LIN {X 0,Y 654.858,Z 275.472,A -85,B 0,C 180,E1 -5918.674,E2 -5918.674} C_VEL
LIN {X 0,Y 654.812,Z 275.476,A -85,B 0,C 180,E1 -5921.282,E2 -5921.282} C_VEL
LIN {X 0,Y 654.839,Z 275.478,A -85,B 0,C 180,E1 -5923.853,E2 -5923.853} C_VEL
LIN {X 0,Y 654.892,Z 275.466,A -85,B 0,C 180,E1 -5927.02,E2 -5927.02} C_VEL
LIN {X 0,Y 654.922,Z 275.602,A -85,B 0,C 180,E1 -5929.598,E2 -5929.598} C_VEL
LIN {X 0,Y 656.022,Z 282.75,A -85,B 0,C 180,E1 -5930.474,E2 -5930.474} C_VEL
LIN {X 0,Y 655.91,Z 303.676,A -85,B 0,C 180,E1 -5932.946,E2 -5932.946} C_VEL
LIN {X 0,Y 655.529,Z 325.625,A -85,B 0,C 180,E1 -5935.557,E2 -5935.557} C_VEL
LIN {X 0,Y 655.353,Z 341.331,A -85,B 0,C 180,E1 -5937.435,E2 -5937.435} C_VEL
LIN {X 0,Y 657.094,Z 353.746,A -85,B 0,C 180,E1 -5937.633,E2 -5937.633} C_VEL
LIN {X 0,Y 656.345,Z 478.954,A -85,B 0,C 180,E1 -5939.083,E2 -5939.083} C_VEL
LIN {X 0,Y 656.153,Z 493.285,A -85,B 0,C 180,E1 -5939.369,E2 -5939.369} C_VEL
LIN {X 0,Y 655.95,Z 507.048,A -85,B 0,C 180,E1 -5939.771,E2 -5939.771} C_VEL
LIN {X 0,Y 655.672,Z 519.008,A -85,B 0,C 180,E1 -5940.23,E2 -5940.23} C_VEL
LIN {X 0,Y 655.42,Z 531.637,A -85,B 0,C 180,E1 -5940.842,E2 -5940.842} C_VEL
LIN {X 0,Y 655.226,Z 543.124,A -85,B 0,C 180,E1 -5941.531,E2 -5941.531} C_VEL
LIN {X 0,Y 654.912,Z 553.719,A -85,B 0,C 180,E1 -5942.299,E2 -5942.299} C_VEL
LIN {X 0,Y 654.674,Z 564.21,A -85,B 0,C 180,E1 -5943.22,E2 -5943.22} C_VEL
LIN {X 0,Y 654.448,Z 572.913,A -85,B 0,C 180,E1 -5944.143,E2 -5944.143} C_VEL
LIN {X 0,Y 654.36,Z 581.161,A -85,B 0,C 180,E1 -5945.208,E2 -5945.208} C_VEL
LIN {X 0,Y 654.28,Z 587.098,A -85,B 0,C 180,E1 -5946.146,E2 -5946.146} C_VEL
LIN {X 0,Y 654.158,Z 593.341,A -85,B 0,C 180,E1 -5947.382,E2 -5947.382} C_VEL
LIN {X 0,Y 654.104,Z 597.95,A -85,B 0,C 180,E1 -5948.622,E2 -5948.622} C_VEL
LIN {X 0,Y 654.115,Z 601.066,A -85,B 0,C 180,E1 -5949.879,E2 -5949.879} C_VEL
LIN {X 0,Y 654.026,Z 602.743,A -85,B 0,C 180,E1 -5951.115,E2 -5951.115} C_VEL
LIN {X 0,Y 654.042,Z 603.068,A -85,B 0,C 180,E1 -5952.368,E2 -5952.368} C_VEL
LIN {X 0,Y 654.063,Z 602.012,A -85,B 0,C 180,E1 -5953.627,E2 -5953.627} C_VEL
LIN {X 0,Y 654.089,Z 599.535,A -85,B 0,C 180,E1 -5954.893,E2 -5954.893} C_VEL
LIN {X 0,Y 654.135,Z 596.647,A -85,B 0,C 180,E1 -5955.846,E2 -5955.846} C_VEL
LIN {X 0,Y 654.194,Z 591.408,A -85,B 0,C 180,E1 -5957.124,E2 -5957.124} C_VEL
LIN {X 0,Y 654.265,Z 586.234,A -85,B 0,C 180,E1 -5958.087,E2 -5958.087} C_VEL
LIN {X 0,Y 654.409,Z 578.75,A -85,B 0,C 180,E1 -5959.216,E2 -5959.216} C_VEL
LIN {X 0,Y 654.569,Z 570.797,A -85,B 0,C 180,E1 -5960.188,E2 -5960.188} C_VEL
LIN {X 0,Y 654.784,Z 561.084,A -85,B 0,C 180,E1 -5961.164,E2 -5961.164} C_VEL
LIN {X 0,Y 655.022,Z 550.211,A -85,B 0,C 180,E1 -5962.062,E2 -5962.062} C_VEL
LIN {X 0,Y 655.346,Z 538.21,A -85,B 0,C 180,E1 -5962.873,E2 -5962.873} C_VEL
LIN {X 0,Y 655.567,Z 526.146,A -85,B 0,C 180,E1 -5963.537,E2 -5963.537} C_VEL
LIN {X 0,Y 655.866,Z 513.079,A -85,B 0,C 180,E1 -5964.111,E2 -5964.111} C_VEL
LIN {X 0,Y 656.125,Z 499.646,A -85,B 0,C 180,E1 -5964.562,E2 -5964.562} C_VEL
LIN {X 0,Y 656.33,Z 485.485,A -85,B 0,C 180,E1 -5964.905,E2 -5964.905} C_VEL
LIN {X 0,Y 656.443,Z 470.534,A -85,B 0,C 180,E1 -5965.135,E2 -5965.135} C_VEL
LIN {X 0,Y 656.965,Z 351.438,A -85,B 0,C 180,E1 -5966.492,E2 -5966.492} C_VEL
LIN {X 0,Y 655.32,Z 341.034,A -85,B 0,C 180,E1 -5966.661,E2 -5966.661} C_VEL
LIN {X 0,Y 655.667,Z 317.93,A -85,B 0,C 180,E1 -5969.465,E2 -5969.465} C_VEL
LIN {X 0,Y 655.064,Z 314.605,A -85,B 0,C 180,E1 -5969.889,E2 -5969.889} C_VEL
LIN {X 0,Y 649.559,Z 304.313,A -85,B 0,C 180,E1 -5971.302,E2 -5971.302} C_VEL
LIN {X 0,Y 649.016,Z 300.937,A -85,B 0,C 180,E1 -5971.729,E2 -5971.729} C_VEL
LIN {X 0,Y 649.167,Z 283.958,A -85,B 0,C 180,E1 -5973.815,E2 -5973.815} C_VEL
LIN {X 0,Y 647.818,Z 276.352,A -85,B 0,C 180,E1 -5974.804,E2 -5974.804} C_VEL
LIN {X 0,Y 647.753,Z 276.352,A -85,B 0,C 180,E1 -5977.269,E2 -5977.269} C_VEL
LIN {X 0,Y 647.771,Z 276.354,A -85,B 0,C 180,E1 -5979.848,E2 -5979.848} C_VEL
LIN {X 0,Y 647.739,Z 276.355,A -85,B 0,C 180,E1 -5982.664,E2 -5982.664} C_VEL
LIN {X 0,Y 647.769,Z 276.352,A -85,B 0,C 180,E1 -5985.342,E2 -5985.342} C_VEL
LIN {X 0,Y 647.733,Z 276.357,A -85,B 0,C 180,E1 -5988.258,E2 -5988.258} C_VEL
LIN {X 0,Y 647.746,Z 276.354,A -85,B 0,C 180,E1 -5990.356,E2 -5990.356} C_VEL
LIN {X 0,Y 647.736,Z 276.355,A -85,B 0,C 180,E1 -5992.729,E2 -5992.729} C_VEL
LIN {X 0,Y 647.769,Z 276.356,A -85,B 0,C 180,E1 -5995.266,E2 -5995.266} C_VEL
LIN {X 0,Y 647.775,Z 276.35,A -85,B 0,C 180,E1 -5998.004,E2 -5998.004} C_VEL
LIN {X 0,Y 647.754,Z 276.353,A -85,B 0,C 180,E1 -6000.17,E2 -6000.17} C_VEL
LIN {X 0,Y 647.796,Z 276.353,A -85,B 0,C 180,E1 -6002.99,E2 -6002.99} C_VEL
LIN {X 0,Y 647.767,Z 276.351,A -85,B 0,C 180,E1 -6005.737,E2 -6005.737} C_VEL
LIN {X 0,Y 647.798,Z 276.353,A -85,B 0,C 180,E1 -6008.429,E2 -6008.429} C_VEL
LIN {X 0,Y 647.806,Z 276.348,A -85,B 0,C 180,E1 -6011.071,E2 -6011.071} C_VEL
LIN {X 0,Y 647.824,Z 276.344,A -85,B 0,C 180,E1 -6013.672,E2 -6013.672} C_VEL
LIN {X 0,Y 647.831,Z 276.35,A -85,B 0,C 180,E1 -6016.238,E2 -6016.238} C_VEL
LIN {X 0,Y 647.825,Z 276.343,A -85,B 0,C 180,E1 -6018.776,E2 -6018.776} C_VEL
LIN {X 0,Y 647.84,Z 276.343,A -85,B 0,C 180,E1 -6020.665,E2 -6020.665} C_VEL
LIN {X 0,Y 647.877,Z 276.339,A -85,B 0,C 180,E1 -6023.169,E2 -6023.169} C_VEL
LIN {X 0,Y 647.905,Z 276.391,A -85,B 0,C 180,E1 -6024.139,E2 -6024.139} C_VEL
LIN {X 0,Y 648.473,Z 281.744,A -85,B 0,C 180,E1 -6025.041,E2 -6025.041} C_VEL
LIN {X 0,Y 648.237,Z 295.521,A -85,B 0,C 180,E1 -6027.289,E2 -6027.289} C_VEL
LIN {X 0,Y 650.27,Z 305.689,A -85,B 0,C 180,E1 -6027.452,E2 -6027.452} C_VEL
LIN {X 0,Y 649.684,Z 431.042,A -85,B 0,C 180,E1 -6028.86,E2 -6028.86} C_VEL
LIN {X 0,Y 649.542,Z 445.303,A -85,B 0,C 180,E1 -6029.149,E2 -6029.149} C_VEL
LIN {X 0,Y 649.298,Z 459.578,A -85,B 0,C 180,E1 -6029.574,E2 -6029.574} C_VEL
LIN {X 0,Y 649.028,Z 472.244,A -85,B 0,C 180,E1 -6030.076,E2 -6030.076} C_VEL
LIN {X 0,Y 648.791,Z 484.553,A -85,B 0,C 180,E1 -6030.694,E2 -6030.694} C_VEL
LIN {X 0,Y 648.467,Z 495.848,A -85,B 0,C 180,E1 -6031.391,E2 -6031.391} C_VEL
LIN {X 0,Y 648.173,Z 506.232,A -85,B 0,C 180,E1 -6032.166,E2 -6032.166} C_VEL
LIN {X 0,Y 647.846,Z 516.572,A -85,B 0,C 180,E1 -6033.097,E2 -6033.097} C_VEL
LIN {X 0,Y 647.639,Z 525.114,A -85,B 0,C 180,E1 -6034.03,E2 -6034.03} C_VEL
LIN {X 0,Y 647.441,Z 533.416,A -85,B 0,C 180,E1 -6035.13,E2 -6035.13} C_VEL
LIN {X 0,Y 647.289,Z 539.975,A -85,B 0,C 180,E1 -6036.211,E2 -6036.211} C_VEL
LIN {X 0,Y 647.229,Z 544.542,A -85,B 0,C 180,E1 -6037.148,E2 -6037.148} C_VEL
LIN {X 0,Y 647.111,Z 548.238,A -85,B 0,C 180,E1 -6038.088,E2 -6038.088} C_VEL
LIN {X 0,Y 647.087,Z 551.85,A -85,B 0,C 180,E1 -6039.343,E2 -6039.343} C_VEL
LIN {X 0,Y 647.054,Z 554.075,A -85,B 0,C 180,E1 -6040.603,E2 -6040.603} C_VEL
LIN {X 0,Y 647.018,Z 554.949,A -85,B 0,C 180,E1 -6041.868,E2 -6041.868} C_VEL
LIN {X 0,Y 647.077,Z 554.469,A -85,B 0,C 180,E1 -6043.138,E2 -6043.138} C_VEL
LIN {X 0,Y 647.031,Z 552.613,A -85,B 0,C 180,E1 -6044.416,E2 -6044.416} C_VEL
LIN {X 0,Y 647.168,Z 549.3,A -85,B 0,C 180,E1 -6045.697,E2 -6045.697} C_VEL
LIN {X 0,Y 647.223,Z 544.379,A -85,B 0,C 180,E1 -6046.988,E2 -6046.988} C_VEL
LIN {X 0,Y 647.321,Z 539.593,A -85,B 0,C 180,E1 -6047.956,E2 -6047.956} C_VEL
LIN {X 0,Y 647.492,Z 532.494,A -85,B 0,C 180,E1 -6049.099,E2 -6049.099} C_VEL
LIN {X 0,Y 647.659,Z 524.764,A -85,B 0,C 180,E1 -6050.11,E2 -6050.11} C_VEL
LIN {X 0,Y 647.94,Z 515.908,A -85,B 0,C 180,E1 -6051.064,E2 -6051.064} C_VEL
LIN {X 0,Y 648.218,Z 505.973,A -85,B 0,C 180,E1 -6051.952,E2 -6051.952} C_VEL
LIN {X 0,Y 648.537,Z 495.768,A -85,B 0,C 180,E1 -6052.711,E2 -6052.711} C_VEL
LIN {X 0,Y 648.837,Z 484.221,A -85,B 0,C 180,E1 -6053.421,E2 -6053.421} C_VEL
LIN {X 0,Y 649.077,Z 471.862,A -85,B 0,C 180,E1 -6054.038,E2 -6054.038} C_VEL
LIN {X 0,Y 649.355,Z 459.191,A -85,B 0,C 180,E1 -6054.536,E2 -6054.536} C_VEL
LIN {X 0,Y 649.544,Z 444.878,A -85,B 0,C 180,E1 -6054.958,E2 -6054.958} C_VEL
LIN {X 0,Y 649.693,Z 430.473,A -85,B 0,C 180,E1 -6055.245,E2 -6055.245} C_VEL
LIN {X 0,Y 650.21,Z 305.17,A -85,B 0,C 180,E1 -6056.654,E2 -6056.654} C_VEL
LIN {X 0,Y 648.261,Z 295.606,A -85,B 0,C 180,E1 -6056.827,E2 -6056.827} C_VEL
LIN {X 0,Y 648.558,Z 281.937,A -85,B 0,C 180,E1 -6059.076,E2 -6059.076} C_VEL
LIN {X 0,Y 647.813,Z 276.353,A -85,B 0,C 180,E1 -6060.056,E2 -6060.056} C_VEL
LIN {X 0,Y 647.739,Z 276.357,A -85,B 0,C 180,E1 -6062.728,E2 -6062.728} C_VEL
LIN {X 0,Y 647.75,Z 276.353,A -85,B 0,C 180,E1 -6064.965,E2 -6064.965} C_VEL
LIN {X 0,Y 647.742,Z 276.359,A -85,B 0,C 180,E1 -6067.871,E2 -6067.871} C_VEL
LIN {X 0,Y 647.74,Z 276.356,A -85,B 0,C 180,E1 -6070.45,E2 -6070.45} C_VEL
LIN {X 0,Y 647.728,Z 276.355,A -85,B 0,C 180,E1 -6072.94,E2 -6072.94} C_VEL
LIN {X 0,Y 647.745,Z 276.35,A -85,B 0,C 180,E1 -6075.533,E2 -6075.533} C_VEL
LIN {X 0,Y 647.762,Z 276.355,A -85,B 0,C 180,E1 -6078.252,E2 -6078.252} C_VEL
LIN {X 0,Y 647.755,Z 276.353,A -85,B 0,C 180,E1 -6080.358,E2 -6080.358} C_VEL
LIN {X 0,Y 647.746,Z 276.35,A -85,B 0,C 180,E1 -6083.146,E2 -6083.146} C_VEL
LIN {X 0,Y 647.747,Z 276.346,A -85,B 0,C 180,E1 -6085.264,E2 -6085.264} C_VEL
LIN {X 0,Y 647.752,Z 276.355,A -85,B 0,C 180,E1 -6088.004,E2 -6088.004} C_VEL
LIN {X 0,Y 647.789,Z 276.349,A -85,B 0,C 180,E1 -6090.172,E2 -6090.172} C_VEL
LIN {X 0,Y 647.769,Z 276.346,A -85,B 0,C 180,E1 -6092.99,E2 -6092.99} C_VEL
LIN {X 0,Y 647.754,Z 276.355,A -85,B 0,C 180,E1 -6095.738,E2 -6095.738} C_VEL
LIN {X 0,Y 647.79,Z 276.345,A -85,B 0,C 180,E1 -6098.413,E2 -6098.413} C_VEL
LIN {X 0,Y 647.777,Z 276.349,A -85,B 0,C 180,E1 -6101.071,E2 -6101.071} C_VEL
LIN {X 0,Y 647.787,Z 276.352,A -85,B 0,C 180,E1 -6103.672,E2 -6103.672} C_VEL
LIN {X 0,Y 647.829,Z 276.338,A -85,B 0,C 180,E1 -6106.669,E2 -6106.669} C_VEL
LIN {X 0,Y 647.805,Z 276.345,A -85,B 0,C 180,E1 -6109.706,E2 -6109.706} C_VEL
LIN {X 0,Y 647.846,Z 276.338,A -85,B 0,C 180,E1 -6112.545,E2 -6112.545} C_VEL
LIN {X 0,Y 647.901,Z 276.339,A -85,B 0,C 180,E1 -6115.038,E2 -6115.038} C_VEL
LIN {X 0,Y 647.945,Z 276.33,A -85,B 0,C 180,E1 -6118.761,E2 -6118.761} C_VEL
LIN {X 0,Y 647.974,Z 276.325,A -85,B 0,C 180,E1 -6121.239,E2 -6121.239} C_VEL
LIN {X 0,Y 647.912,Z 276.34,A -85,B 0,C 180,E1 -6124.962,E2 -6124.962} C_VEL
LIN {X 0,Y 647.849,Z 276.337,A -85,B 0,C 180,E1 -6127.455,E2 -6127.455} C_VEL
LIN {X 0,Y 647.85,Z 276.342,A -85,B 0,C 180,E1 -6130.591,E2 -6130.591} C_VEL
LIN {X 0,Y 647.829,Z 276.341,A -85,B 0,C 180,E1 -6133.331,E2 -6133.331} C_VEL
LIN {X 0,Y 647.801,Z 276.346,A -85,B 0,C 180,E1 -6136.328,E2 -6136.328} C_VEL
LIN {X 0,Y 647.787,Z 276.344,A -85,B 0,C 180,E1 -6138.275,E2 -6138.275} C_VEL
LIN {X 0,Y 647.788,Z 276.348,A -85,B 0,C 180,E1 -6140.244,E2 -6140.244} C_VEL
LIN {X 0,Y 647.782,Z 276.352,A -85,B 0,C 180,E1 -6142.909,E2 -6142.909} C_VEL
LIN {X 0,Y 647.725,Z 276.352,A -85,B 0,C 180,E1 -6145.63,E2 -6145.63} C_VEL
LIN {X 0,Y 647.761,Z 276.348,A -85,B 0,C 180,E1 -6147.708,E2 -6147.708} C_VEL
LIN {X 0,Y 647.781,Z 276.35,A -85,B 0,C 180,E1 -6150.118,E2 -6150.118} C_VEL
LIN {X 0,Y 647.766,Z 276.354,A -85,B 0,C 180,E1 -6152.729,E2 -6152.729} C_VEL
LIN {X 0,Y 647.779,Z 276.34,A -85,B 0,C 180,E1 -6154.966,E2 -6154.966} C_VEL
LIN {X 0,Y 647.756,Z 276.347,A -85,B 0,C 180,E1 -6157.269,E2 -6157.269} C_VEL
LIN {X 0,Y 647.782,Z 276.35,A -85,B 0,C 180,E1 -6159.854,E2 -6159.854} C_VEL
LIN {X 0,Y 647.771,Z 276.356,A -85,B 0,C 180,E1 -6162.099,E2 -6162.099} C_VEL
LIN {X 0,Y 647.772,Z 276.35,A -85,B 0,C 180,E1 -6164.656,E2 -6164.656} C_VEL
LIN {X 0,Y 647.782,Z 276.346,A -85,B 0,C 180,E1 -6167.331,E2 -6167.331} C_VEL
LIN {X 0,Y 647.798,Z 276.346,A -85,B 0,C 180,E1 -6169.554,E2 -6169.554} C_VEL
LIN {X 0,Y 647.775,Z 276.358,A -85,B 0,C 180,E1 -6172.125,E2 -6172.125} C_VEL
LIN {X 0,Y 647.82,Z 276.352,A -85,B 0,C 180,E1 -6174.28,E2 -6174.28} C_VEL
LIN {X 0,Y 647.778,Z 276.353,A -85,B 0,C 180,E1 -6176.535,E2 -6176.535} C_VEL
LIN {X 0,Y 647.791,Z 276.35,A -85,B 0,C 180,E1 -6178.736,E2 -6178.736} C_VEL
LIN {X 0,Y 647.813,Z 276.346,A -85,B 0,C 180,E1 -6181.141,E2 -6181.141} C_VEL
LIN {X 0,Y 647.759,Z 276.358,A -85,B 0,C 180,E1 -6183.833,E2 -6183.833} C_VEL
LIN {X 0,Y 647.808,Z 276.453,A -85,B 0,C 180,E1 -6184.933,E2 -6184.933} C_VEL
LIN {X 0,Y 649.955,Z 287.8,A -85,B 0,C 180,E1 -6186.352,E2 -6186.352} C_VEL
LIN {X 0,Y 649.394,Z 310.669,A -85,B 0,C 180,E1 -6188.985,E2 -6188.985} C_VEL
LIN {X 0,Y 648.728,Z 336.782,A -85,B 0,C 180,E1 -6191.936,E2 -6191.936} C_VEL
LIN {X 0,Y 648.218,Z 362.614,A -85,B 0,C 180,E1 -6194.811,E2 -6194.811} C_VEL
LIN {X 0,Y 648.158,Z 366.227,A -85,B 0,C 180,E1 -6195.21,E2 -6195.21} C_VEL
LIN {X 0,Y 650.159,Z 382.238,A -85,B 0,C 180,E1 -6195.436,E2 -6195.436} C_VEL
LIN {X 0,Y 649.597,Z 503.865,A -85,B 0,C 180,E1 -6196.795,E2 -6196.795} C_VEL
LIN {X 0,Y 649.346,Z 517.951,A -85,B 0,C 180,E1 -6197.068,E2 -6197.068} C_VEL
LIN {X 0,Y 649.084,Z 531.649,A -85,B 0,C 180,E1 -6197.459,E2 -6197.459} C_VEL
LIN {X 0,Y 648.782,Z 544.087,A -85,B 0,C 180,E1 -6197.928,E2 -6197.928} C_VEL
LIN {X 0,Y 648.407,Z 557.099,A -85,B 0,C 180,E1 -6198.553,E2 -6198.553} C_VEL
LIN {X 0,Y 648.165,Z 568.915,A -85,B 0,C 180,E1 -6199.258,E2 -6199.258} C_VEL
LIN {X 0,Y 647.896,Z 579.737,A -85,B 0,C 180,E1 -6200.041,E2 -6200.041} C_VEL
LIN {X 0,Y 647.591,Z 590.455,A -85,B 0,C 180,E1 -6200.978,E2 -6200.978} C_VEL
LIN {X 0,Y 647.373,Z 599.315,A -85,B 0,C 180,E1 -6201.916,E2 -6201.916} C_VEL
LIN {X 0,Y 647.247,Z 607.826,A -85,B 0,C 180,E1 -6203.009,E2 -6203.009} C_VEL
LIN {X 0,Y 647.127,Z 614.684,A -85,B 0,C 180,E1 -6204.1,E2 -6204.1} C_VEL
LIN {X 0,Y 647.079,Z 620.81,A -85,B 0,C 180,E1 -6205.345,E2 -6205.345} C_VEL
LIN {X 0,Y 647.029,Z 624.325,A -85,B 0,C 180,E1 -6206.277,E2 -6206.277} C_VEL
LIN {X 0,Y 647.083,Z 627.745,A -85,B 0,C 180,E1 -6207.52,E2 -6207.52} C_VEL
LIN {X 0,Y 647.049,Z 629.762,A -85,B 0,C 180,E1 -6208.761,E2 -6208.761} C_VEL
LIN {X 0,Y 647.02,Z 630.43,A -85,B 0,C 180,E1 -6210.002,E2 -6210.002} C_VEL
LIN {X 0,Y 647.049,Z 629.765,A -85,B 0,C 180,E1 -6211.242,E2 -6211.242} C_VEL
LIN {X 0,Y 647.084,Z 627.752,A -85,B 0,C 180,E1 -6212.483,E2 -6212.483} C_VEL
LIN {X 0,Y 647.029,Z 624.339,A -85,B 0,C 180,E1 -6213.726,E2 -6213.726} C_VEL
LIN {X 0,Y 647.08,Z 620.834,A -85,B 0,C 180,E1 -6214.658,E2 -6214.658} C_VEL
LIN {X 0,Y 647.134,Z 616.381,A -85,B 0,C 180,E1 -6215.592,E2 -6215.592} C_VEL
LIN {X 0,Y 647.2,Z 609.95,A -85,B 0,C 180,E1 -6216.683,E2 -6216.683} C_VEL
LIN {X 0,Y 647.352,Z 601.971,A -85,B 0,C 180,E1 -6217.775,E2 -6217.775} C_VEL
LIN {X 0,Y 647.536,Z 593.636,A -85,B 0,C 180,E1 -6218.712,E2 -6218.712} C_VEL
LIN {X 0,Y 647.759,Z 583.61,A -85,B 0,C 180,E1 -6219.65,E2 -6219.65} C_VEL
LIN {X 0,Y 648.055,Z 572.845,A -85,B 0,C 180,E1 -6220.483,E2 -6220.483} C_VEL
LIN {X 0,Y 648.309,Z 561.398,A -85,B 0,C 180,E1 -6221.215,E2 -6221.215} C_VEL
LIN {X 0,Y 648.658,Z 549.41,A -85,B 0,C 180,E1 -6221.841,E2 -6221.841} C_VEL
LIN {X 0,Y 648.976,Z 536.202,A -85,B 0,C 180,E1 -6222.388,E2 -6222.388} C_VEL
LIN {X 0,Y 649.237,Z 522.519,A -85,B 0,C 180,E1 -6222.819,E2 -6222.819} C_VEL
LIN {X 0,Y 649.511,Z 508.407,A -85,B 0,C 180,E1 -6223.13,E2 -6223.13} C_VEL
LIN {X 0,Y 649.71,Z 490.629,A -85,B 0,C 180,E1 -6223.364,E2 -6223.364} C_VEL
LIN {X 0,Y 650.01,Z 380.445,A -85,B 0,C 180,E1 -6224.587,E2 -6224.587} C_VEL
LIN {X 0,Y 648.178,Z 366.315,A -85,B 0,C 180,E1 -6224.793,E2 -6224.793} C_VEL
LIN {X 0,Y 648.534,Z 343.886,A -85,B 0,C 180,E1 -6227.279,E2 -6227.279} C_VEL
LIN {X 0,Y 648.95,Z 325.006,A -85,B 0,C 180,E1 -6229.385,E2 -6229.385} C_VEL
LIN {X 0,Y 649.466,Z 305.113,A -85,B 0,C 180,E1 -6231.628,E2 -6231.628} C_VEL
LIN {X 0,Y 649.889,Z 287.5,A -85,B 0,C 180,E1 -6233.634,E2 -6233.634} C_VEL
LIN {X 0,Y 647.815,Z 276.349,A -85,B 0,C 180,E1 -6235.006,E2 -6235.006} C_VEL
LIN {X 0,Y 647.779,Z 276.356,A -85,B 0,C 180,E1 -6237.709,E2 -6237.709} C_VEL
LIN {X 0,Y 647.743,Z 276.358,A -85,B 0,C 180,E1 -6240.107,E2 -6240.107} C_VEL
LIN {X 0,Y 647.749,Z 276.351,A -85,B 0,C 180,E1 -6242.731,E2 -6242.731} C_VEL
LIN {X 0,Y 647.759,Z 276.352,A -85,B 0,C 180,E1 -6244.968,E2 -6244.968} C_VEL
LIN {X 0,Y 647.738,Z 276.359,A -85,B 0,C 180,E1 -6247.271,E2 -6247.271} C_VEL
LIN {X 0,Y 647.758,Z 276.354,A -85,B 0,C 180,E1 -6249.848,E2 -6249.848} C_VEL
LIN {X 0,Y 647.729,Z 276.355,A -85,B 0,C 180,E1 -6252.664,E2 -6252.664} C_VEL
LIN {X 0,Y 647.757,Z 276.355,A -85,B 0,C 180,E1 -6255.537,E2 -6255.537} C_VEL
LIN {X 0,Y 647.736,Z 276.353,A -85,B 0,C 180,E1 -6258.259,E2 -6258.259} C_VEL
LIN {X 0,Y 647.749,Z 276.353,A -85,B 0,C 180,E1 -6260.357,E2 -6260.357} C_VEL
LIN {X 0,Y 647.745,Z 276.358,A -85,B 0,C 180,E1 -6263.151,E2 -6263.151} C_VEL
LIN {X 0,Y 647.776,Z 276.35,A -85,B 0,C 180,E1 -6265.266,E2 -6265.266} C_VEL
LIN {X 0,Y 647.775,Z 276.35,A -85,B 0,C 180,E1 -6268.005,E2 -6268.005} C_VEL
LIN {X 0,Y 647.774,Z 276.354,A -85,B 0,C 180,E1 -6270.172,E2 -6270.172} C_VEL
LIN {X 0,Y 647.771,Z 276.351,A -85,B 0,C 180,E1 -6272.99,E2 -6272.99} C_VEL
LIN {X 0,Y 647.769,Z 276.353,A -85,B 0,C 180,E1 -6275.739,E2 -6275.739} C_VEL
LIN {X 0,Y 647.8,Z 276.355,A -85,B 0,C 180,E1 -6278.43,E2 -6278.43} C_VEL
LIN {X 0,Y 647.792,Z 276.35,A -85,B 0,C 180,E1 -6281.072,E2 -6281.072} C_VEL
LIN {X 0,Y 647.804,Z 276.353,A -85,B 0,C 180,E1 -6283.672,E2 -6283.672} C_VEL
LIN {X 0,Y 647.829,Z 276.345,A -85,B 0,C 180,E1 -6286.682,E2 -6286.682} C_VEL
LIN {X 0,Y 647.857,Z 276.444,A -85,B 0,C 180,E1 -6289.473,E2 -6289.473} C_VEL
LIN {X 0,Y 649.059,Z 283.7,A -85,B 0,C 180,E1 -6290.371,E2 -6290.371} C_VEL
LIN {X 0,Y 648.955,Z 304.702,A -85,B 0,C 180,E1 -6292.87,E2 -6292.87} C_VEL
LIN {X 0,Y 648.543,Z 326.809,A -85,B 0,C 180,E1 -6295.509,E2 -6295.509} C_VEL
LIN {X 0,Y 648.393,Z 341.466,A -85,B 0,C 180,E1 -6297.272,E2 -6297.272} C_VEL
LIN {X 0,Y 650.215,Z 353.505,A -85,B 0,C 180,E1 -6297.472,E2 -6297.472} C_VEL
LIN {X 0,Y 649.407,Z 479.295,A -85,B 0,C 180,E1 -6298.957,E2 -6298.957} C_VEL
LIN {X 0,Y 649.224,Z 493.533,A -85,B 0,C 180,E1 -6299.247,E2 -6299.247} C_VEL
LIN {X 0,Y 649,Z 507.262,A -85,B 0,C 180,E1 -6299.652,E2 -6299.652} C_VEL
LIN {X 0,Y 648.659,Z 520.086,A -85,B 0,C 180,E1 -6300.155,E2 -6300.155} C_VEL
LIN {X 0,Y 648.409,Z 532.508,A -85,B 0,C 180,E1 -6300.774,E2 -6300.774} C_VEL
LIN {X 0,Y 648.212,Z 544.992,A -85,B 0,C 180,E1 -6301.548,E2 -6301.548} C_VEL
LIN {X 0,Y 647.845,Z 555.319,A -85,B 0,C 180,E1 -6302.324,E2 -6302.324} C_VEL
LIN {X 0,Y 647.629,Z 565.577,A -85,B 0,C 180,E1 -6303.255,E2 -6303.255} C_VEL
LIN {X 0,Y 647.351,Z 574.096,A -85,B 0,C 180,E1 -6304.188,E2 -6304.188} C_VEL
LIN {X 0,Y 647.284,Z 581.483,A -85,B 0,C 180,E1 -6305.167,E2 -6305.167} C_VEL
LIN {X 0,Y 647.177,Z 587.955,A -85,B 0,C 180,E1 -6306.213,E2 -6306.213} C_VEL
LIN {X 0,Y 647.085,Z 592.645,A -85,B 0,C 180,E1 -6307.151,E2 -6307.151} C_VEL
LIN {X 0,Y 647.028,Z 597.491,A -85,B 0,C 180,E1 -6308.404,E2 -6308.404} C_VEL
LIN {X 0,Y 647.01,Z 600.115,A -85,B 0,C 180,E1 -6309.346,E2 -6309.346} C_VEL
LIN {X 0,Y 646.95,Z 602.376,A -85,B 0,C 180,E1 -6310.606,E2 -6310.606} C_VEL
LIN {X 0,Y 646.938,Z 603.256,A -85,B 0,C 180,E1 -6311.871,E2 -6311.871} C_VEL
LIN {X 0,Y 647.003,Z 602.753,A -85,B 0,C 180,E1 -6313.141,E2 -6313.141} C_VEL
LIN {X 0,Y 646.94,Z 600.831,A -85,B 0,C 180,E1 -6314.42,E2 -6314.42} C_VEL
LIN {X 0,Y 647.035,Z 597.395,A -85,B 0,C 180,E1 -6315.702,E2 -6315.702} C_VEL
LIN {X 0,Y 647.109,Z 592.357,A -85,B 0,C 180,E1 -6316.993,E2 -6316.993} C_VEL
LIN {X 0,Y 647.181,Z 587.523,A -85,B 0,C 180,E1 -6317.944,E2 -6317.944} C_VEL
LIN {X 0,Y 647.333,Z 580.148,A -85,B 0,C 180,E1 -6319.106,E2 -6319.106} C_VEL
LIN {X 0,Y 647.493,Z 572.322,A -85,B 0,C 180,E1 -6320.104,E2 -6320.104} C_VEL
LIN {X 0,Y 647.697,Z 563.116,A -85,B 0,C 180,E1 -6321.074,E2 -6321.074} C_VEL
LIN {X 0,Y 647.981,Z 552.712,A -85,B 0,C 180,E1 -6321.98,E2 -6321.98} C_VEL
LIN {X 0,Y 648.281,Z 541.099,A -85,B 0,C 180,E1 -6322.806,E2 -6322.806} C_VEL
LIN {X 0,Y 648.554,Z 528.145,A -85,B 0,C 180,E1 -6323.553,E2 -6323.553} C_VEL
LIN {X 0,Y 648.846,Z 515.544,A -85,B 0,C 180,E1 -6324.134,E2 -6324.134} C_VEL
LIN {X 0,Y 649.122,Z 502.908,A -85,B 0,C 180,E1 -6324.59,E2 -6324.59} C_VEL
LIN {X 0,Y 649.335,Z 488.251,A -85,B 0,C 180,E1 -6324.981,E2 -6324.981} C_VEL
LIN {X 0,Y 649.486,Z 473.738,A -85,B 0,C 180,E1 -6325.23,E2 -6325.23} C_VEL
LIN {X 0,Y 650.104,Z 352.375,A -85,B 0,C 180,E1 -6326.633,E2 -6326.633} C_VEL
LIN {X 0,Y 648.297,Z 341.19,A -85,B 0,C 180,E1 -6326.81,E2 -6326.81} C_VEL
LIN {X 0,Y 648.7,Z 318.347,A -85,B 0,C 180,E1 -6329.603,E2 -6329.603} C_VEL
LIN {X 0,Y 649.016,Z 300.937,A -85,B 0,C 180,E1 -6331.729,E2 -6331.729} C_VEL
LIN {X 0,Y 648.543,Z 297.612,A -85,B 0,C 180,E1 -6332.155,E2 -6332.155} C_VEL
LIN {X 0,Y 646.029,Z 292.413,A -85,B 0,C 180,E1 -6332.867,E2 -6332.867} C_VEL
LIN {X 0,Y 642.671,Z 286.255,A -85,B 0,C 180,E1 -6333.731,E2 -6333.731} C_VEL
LIN {X 0,Y 642.044,Z 284.037,A -85,B 0,C 180,E1 -6334.022,E2 -6334.022} C_VEL
LIN {X 0,Y 640.76,Z 277.23,A -85,B 0,C 180,E1 -6334.928,E2 -6334.928} C_VEL
LIN {X 0,Y 640.732,Z 277.23,A -85,B 0,C 180,E1 -6337.748,E2 -6337.748} C_VEL
LIN {X 0,Y 640.727,Z 277.235,A -85,B 0,C 180,E1 -6340.165,E2 -6340.165} C_VEL
LIN {X 0,Y 640.72,Z 277.228,A -85,B 0,C 180,E1 -6342.906,E2 -6342.906} C_VEL
LIN {X 0,Y 640.725,Z 277.232,A -85,B 0,C 180,E1 -6345.6,E2 -6345.6} C_VEL
LIN {X 0,Y 640.685,Z 277.236,A -85,B 0,C 180,E1 -6348.171,E2 -6348.171} C_VEL
LIN {X 0,Y 640.69,Z 277.232,A -85,B 0,C 180,E1 -6350.646,E2 -6350.646} C_VEL
LIN {X 0,Y 640.714,Z 277.233,A -85,B 0,C 180,E1 -6353.038,E2 -6353.038} C_VEL
LIN {X 0,Y 640.716,Z 277.234,A -85,B 0,C 180,E1 -6355.355,E2 -6355.355} C_VEL
LIN {X 0,Y 640.726,Z 277.232,A -85,B 0,C 180,E1 -6357.609,E2 -6357.609} C_VEL
LIN {X 0,Y 640.722,Z 277.23,A -85,B 0,C 180,E1 -6359.808,E2 -6359.808} C_VEL
LIN {X 0,Y 640.74,Z 277.228,A -85,B 0,C 180,E1 -6362.31,E2 -6362.31} C_VEL
LIN {X 0,Y 640.759,Z 277.229,A -85,B 0,C 180,E1 -6365.137,E2 -6365.137} C_VEL
LIN {X 0,Y 640.741,Z 277.226,A -85,B 0,C 180,E1 -6367.503,E2 -6367.503} C_VEL
LIN {X 0,Y 640.786,Z 277.224,A -85,B 0,C 180,E1 -6370.191,E2 -6370.191} C_VEL
LIN {X 0,Y 640.768,Z 277.226,A -85,B 0,C 180,E1 -6372.832,E2 -6372.832} C_VEL
LIN {X 0,Y 640.785,Z 277.223,A -85,B 0,C 180,E1 -6374.789,E2 -6374.789} C_VEL
LIN {X 0,Y 640.783,Z 277.22,A -85,B 0,C 180,E1 -6377.371,E2 -6377.371} C_VEL
LIN {X 0,Y 640.815,Z 277.224,A -85,B 0,C 180,E1 -6379.926,E2 -6379.926} C_VEL
LIN {X 0,Y 640.827,Z 277.219,A -85,B 0,C 180,E1 -6382.462,E2 -6382.462} C_VEL
LIN {X 0,Y 640.874,Z 277.238,A -85,B 0,C 180,E1 -6384.036,E2 -6384.036} C_VEL
LIN {X 0,Y 641.484,Z 282.839,A -85,B 0,C 180,E1 -6384.987,E2 -6384.987} C_VEL
LIN {X 0,Y 641.239,Z 295.858,A -85,B 0,C 180,E1 -6387.122,E2 -6387.122} C_VEL
LIN {X 0,Y 643.449,Z 306.862,A -85,B 0,C 180,E1 -6387.308,E2 -6387.308} C_VEL
LIN {X 0,Y 642.791,Z 430.913,A -85,B 0,C 180,E1 -6388.711,E2 -6388.711} C_VEL
LIN {X 0,Y 642.658,Z 445.356,A -85,B 0,C 180,E1 -6389.003,E2 -6389.003} C_VEL
LIN {X 0,Y 642.423,Z 459.171,A -85,B 0,C 180,E1 -6389.413,E2 -6389.413} C_VEL
LIN {X 0,Y 642.118,Z 472.032,A -85,B 0,C 180,E1 -6389.92,E2 -6389.92} C_VEL
LIN {X 0,Y 641.841,Z 484.477,A -85,B 0,C 180,E1 -6390.546,E2 -6390.546} C_VEL
LIN {X 0,Y 641.508,Z 495.862,A -85,B 0,C 180,E1 -6391.25,E2 -6391.25} C_VEL
LIN {X 0,Y 641.205,Z 506.31,A -85,B 0,C 180,E1 -6392.033,E2 -6392.033} C_VEL
LIN {X 0,Y 640.846,Z 516.711,A -85,B 0,C 180,E1 -6392.974,E2 -6392.974} C_VEL
LIN {X 0,Y 640.627,Z 525.3,A -85,B 0,C 180,E1 -6393.917,E2 -6393.917} C_VEL
LIN {X 0,Y 640.391,Z 533.573,A -85,B 0,C 180,E1 -6395.018,E2 -6395.018} C_VEL
LIN {X 0,Y 640.285,Z 539.346,A -85,B 0,C 180,E1 -6395.964,E2 -6395.964} C_VEL
LIN {X 0,Y 640.157,Z 545.542,A -85,B 0,C 180,E1 -6397.227,E2 -6397.227} C_VEL
LIN {X 0,Y 640.027,Z 549.09,A -85,B 0,C 180,E1 -6398.178,E2 -6398.178} C_VEL
LIN {X 0,Y 640.006,Z 552.562,A -85,B 0,C 180,E1 -6399.447,E2 -6399.447} C_VEL
LIN {X 0,Y 639.967,Z 554.653,A -85,B 0,C 180,E1 -6400.721,E2 -6400.721} C_VEL
LIN {X 0,Y 639.952,Z 555.394,A -85,B 0,C 180,E1 -6402.001,E2 -6402.001} C_VEL
LIN {X 0,Y 639.981,Z 554.77,A -85,B 0,C 180,E1 -6403.286,E2 -6403.286} C_VEL
LIN {X 0,Y 639.959,Z 552.744,A -85,B 0,C 180,E1 -6404.579,E2 -6404.579} C_VEL
LIN {X 0,Y 640.099,Z 549.255,A -85,B 0,C 180,E1 -6405.875,E2 -6405.875} C_VEL
LIN {X 0,Y 640.181,Z 544.18,A -85,B 0,C 180,E1 -6407.181,E2 -6407.181} C_VEL
LIN {X 0,Y 640.3,Z 539.205,A -85,B 0,C 180,E1 -6408.164,E2 -6408.164} C_VEL
LIN {X 0,Y 640.484,Z 531.946,A -85,B 0,C 180,E1 -6409.317,E2 -6409.317} C_VEL
LIN {X 0,Y 640.723,Z 524.401,A -85,B 0,C 180,E1 -6410.291,E2 -6410.291} C_VEL
LIN {X 0,Y 640.979,Z 514.911,A -85,B 0,C 180,E1 -6411.304,E2 -6411.304} C_VEL
LIN {X 0,Y 641.318,Z 504.491,A -85,B 0,C 180,E1 -6412.218,E2 -6412.218} C_VEL
LIN {X 0,Y 641.649,Z 492.904,A -85,B 0,C 180,E1 -6413.053,E2 -6413.053} C_VEL
LIN {X 0,Y 641.94,Z 479.857,A -85,B 0,C 180,E1 -6413.809,E2 -6413.809} C_VEL
LIN {X 0,Y 642.269,Z 467.082,A -85,B 0,C 180,E1 -6414.395,E2 -6414.395} C_VEL
LIN {X 0,Y 642.578,Z 452.759,A -85,B 0,C 180,E1 -6414.898,E2 -6414.898} C_VEL
LIN {X 0,Y 642.741,Z 438.589,A -85,B 0,C 180,E1 -6415.255,E2 -6415.255} C_VEL
LIN {X 0,Y 642.83,Z 425.311,A -85,B 0,C 180,E1 -6415.469,E2 -6415.469} C_VEL
LIN {X 0,Y 643.409,Z 306.285,A -85,B 0,C 180,E1 -6416.81,E2 -6416.81} C_VEL
LIN {X 0,Y 641.319,Z 296.072,A -85,B 0,C 180,E1 -6416.993,E2 -6416.993} C_VEL
LIN {X 0,Y 641.594,Z 283.059,A -85,B 0,C 180,E1 -6419.146,E2 -6419.146} C_VEL
LIN {X 0,Y 640.737,Z 277.234,A -85,B 0,C 180,E1 -6420.187,E2 -6420.187} C_VEL
LIN {X 0,Y 640.716,Z 277.233,A -85,B 0,C 180,E1 -6422.671,E2 -6422.671} C_VEL
LIN {X 0,Y 640.708,Z 277.23,A -85,B 0,C 180,E1 -6425.407,E2 -6425.407} C_VEL
LIN {X 0,Y 640.696,Z 277.238,A -85,B 0,C 180,E1 -6428.081,E2 -6428.081} C_VEL
LIN {X 0,Y 640.69,Z 277.23,A -85,B 0,C 180,E1 -6430.99,E2 -6430.99} C_VEL
LIN {X 0,Y 640.696,Z 277.238,A -85,B 0,C 180,E1 -6433.817,E2 -6433.817} C_VEL
LIN {X 0,Y 640.714,Z 277.231,A -85,B 0,C 180,E1 -6436.47,E2 -6436.47} C_VEL
LIN {X 0,Y 640.717,Z 277.227,A -85,B 0,C 180,E1 -6439.01,E2 -6439.01} C_VEL
LIN {X 0,Y 640.692,Z 277.238,A -85,B 0,C 180,E1 -6441.916,E2 -6441.916} C_VEL
LIN {X 0,Y 640.738,Z 277.217,A -85,B 0,C 180,E1 -6444.593,E2 -6444.593} C_VEL
LIN {X 0,Y 640.709,Z 277.231,A -85,B 0,C 180,E1 -6447.325,E2 -6447.325} C_VEL
LIN {X 0,Y 640.745,Z 277.232,A -85,B 0,C 180,E1 -6449.811,E2 -6449.811} C_VEL
LIN {X 0,Y 640.741,Z 277.222,A -85,B 0,C 180,E1 -6452.305,E2 -6452.305} C_VEL
LIN {X 0,Y 640.735,Z 277.228,A -85,B 0,C 180,E1 -6455.136,E2 -6455.136} C_VEL
LIN {X 0,Y 640.718,Z 277.232,A -85,B 0,C 180,E1 -6457.504,E2 -6457.504} C_VEL
LIN {X 0,Y 640.756,Z 277.22,A -85,B 0,C 180,E1 -6460.191,E2 -6460.191} C_VEL
LIN {X 0,Y 640.725,Z 277.226,A -85,B 0,C 180,E1 -6462.833,E2 -6462.833} C_VEL
LIN {X 0,Y 640.751,Z 277.223,A -85,B 0,C 180,E1 -6464.79,E2 -6464.79} C_VEL
LIN {X 0,Y 640.768,Z 277.228,A -85,B 0,C 180,E1 -6467.372,E2 -6467.372} C_VEL
LIN {X 0,Y 640.765,Z 277.219,A -85,B 0,C 180,E1 -6469.927,E2 -6469.927} C_VEL
LIN {X 0,Y 640.811,Z 277.213,A -85,B 0,C 180,E1 -6472.463,E2 -6472.463} C_VEL
LIN {X 0,Y 640.852,Z 277.216,A -85,B 0,C 180,E1 -6474.984,E2 -6474.984} C_VEL
LIN {X 0,Y 640.911,Z 277.206,A -85,B 0,C 180,E1 -6478.748,E2 -6478.748} C_VEL
LIN {X 0,Y 640.938,Z 277.201,A -85,B 0,C 180,E1 -6481.252,E2 -6481.252} C_VEL
LIN {X 0,Y 640.865,Z 277.218,A -85,B 0,C 180,E1 -6485.016,E2 -6485.016} C_VEL
LIN {X 0,Y 640.813,Z 277.212,A -85,B 0,C 180,E1 -6487.537,E2 -6487.537} C_VEL
LIN {X 0,Y 640.823,Z 277.215,A -85,B 0,C 180,E1 -6490.362,E2 -6490.362} C_VEL
LIN {X 0,Y 640.784,Z 277.218,A -85,B 0,C 180,E1 -6493.389,E2 -6493.389} C_VEL
LIN {X 0,Y 640.778,Z 277.217,A -85,B 0,C 180,E1 -6495.867,E2 -6495.867} C_VEL
LIN {X 0,Y 640.74,Z 277.225,A -85,B 0,C 180,E1 -6498.483,E2 -6498.483} C_VEL
LIN {X 0,Y 640.729,Z 277.231,A -85,B 0,C 180,E1 -6500.477,E2 -6500.477} C_VEL
LIN {X 0,Y 640.771,Z 277.222,A -85,B 0,C 180,E1 -6503.174,E2 -6503.174} C_VEL
LIN {X 0,Y 640.678,Z 277.231,A -85,B 0,C 180,E1 -6505.933,E2 -6505.933} C_VEL
LIN {X 0,Y 640.758,Z 277.228,A -85,B 0,C 180,E1 -6508.75,E2 -6508.75} C_VEL
LIN {X 0,Y 640.738,Z 277.223,A -85,B 0,C 180,E1 -6511.5,E2 -6511.5} C_VEL
LIN {X 0,Y 640.714,Z 277.228,A -85,B 0,C 180,E1 -6513.886,E2 -6513.886} C_VEL
LIN {X 0,Y 640.753,Z 277.218,A -85,B 0,C 180,E1 -6516.179,E2 -6516.179} C_VEL
LIN {X 0,Y 640.745,Z 277.231,A -85,B 0,C 180,E1 -6518.544,E2 -6518.544} C_VEL
LIN {X 0,Y 640.744,Z 277.224,A -85,B 0,C 180,E1 -6521.04,E2 -6521.04} C_VEL
LIN {X 0,Y 640.74,Z 277.224,A -85,B 0,C 180,E1 -6523.528,E2 -6523.528} C_VEL
LIN {X 0,Y 640.745,Z 277.229,A -85,B 0,C 180,E1 -6526.476,E2 -6526.476} C_VEL
LIN {X 0,Y 640.763,Z 277.221,A -85,B 0,C 180,E1 -6529.016,E2 -6529.016} C_VEL
LIN {X 0,Y 640.739,Z 277.232,A -85,B 0,C 180,E1 -6531.915,E2 -6531.915} C_VEL
LIN {X 0,Y 640.768,Z 277.226,A -85,B 0,C 180,E1 -6534.597,E2 -6534.597} C_VEL
LIN {X 0,Y 640.732,Z 277.233,A -85,B 0,C 180,E1 -6537.613,E2 -6537.613} C_VEL
LIN {X 0,Y 640.764,Z 277.225,A -85,B 0,C 180,E1 -6540.536,E2 -6540.536} C_VEL
LIN {X 0,Y 640.73,Z 277.229,A -85,B 0,C 180,E1 -6542.67,E2 -6542.67} C_VEL
LIN {X 0,Y 640.77,Z 277.328,A -85,B 0,C 180,E1 -6544.768,E2 -6544.768} C_VEL
LIN {X 0,Y 643.032,Z 288.855,A -85,B 0,C 180,E1 -6546.234,E2 -6546.234} C_VEL
LIN {X 0,Y 642.499,Z 308.958,A -85,B 0,C 180,E1 -6548.581,E2 -6548.581} C_VEL
LIN {X 0,Y 641.817,Z 334.849,A -85,B 0,C 180,E1 -6551.551,E2 -6551.551} C_VEL
LIN {X 0,Y 641.23,Z 362.234,A -85,B 0,C 180,E1 -6554.641,E2 -6554.641} C_VEL
LIN {X 0,Y 641.112,Z 365.653,A -85,B 0,C 180,E1 -6555.023,E2 -6555.023} C_VEL
LIN {X 0,Y 643.299,Z 382.12,A -85,B 0,C 180,E1 -6555.277,E2 -6555.277} C_VEL
LIN {X 0,Y 642.706,Z 503.546,A -85,B 0,C 180,E1 -6556.651,E2 -6556.651} C_VEL
LIN {X 0,Y 642.415,Z 517.576,A -85,B 0,C 180,E1 -6556.926,E2 -6556.926} C_VEL
LIN {X 0,Y 642.141,Z 531.261,A -85,B 0,C 180,E1 -6557.321,E2 -6557.321} C_VEL
LIN {X 0,Y 641.832,Z 543.687,A -85,B 0,C 180,E1 -6557.795,E2 -6557.795} C_VEL
LIN {X 0,Y 641.429,Z 556.689,A -85,B 0,C 180,E1 -6558.426,E2 -6558.426} C_VEL
LIN {X 0,Y 641.167,Z 568.497,A -85,B 0,C 180,E1 -6559.14,E2 -6559.14} C_VEL
LIN {X 0,Y 640.863,Z 579.313,A -85,B 0,C 180,E1 -6559.93,E2 -6559.93} C_VEL
LIN {X 0,Y 640.551,Z 590.029,A -85,B 0,C 180,E1 -6560.878,E2 -6560.878} C_VEL
LIN {X 0,Y 640.299,Z 598.889,A -85,B 0,C 180,E1 -6561.826,E2 -6561.826} C_VEL
LIN {X 0,Y 640.158,Z 607.401,A -85,B 0,C 180,E1 -6562.931,E2 -6562.931} C_VEL
LIN {X 0,Y 640.035,Z 614.261,A -85,B 0,C 180,E1 -6564.034,E2 -6564.034} C_VEL
LIN {X 0,Y 639.99,Z 618.993,A -85,B 0,C 180,E1 -6564.979,E2 -6564.979} C_VEL
LIN {X 0,Y 639.955,Z 623.909,A -85,B 0,C 180,E1 -6566.236,E2 -6566.236} C_VEL
LIN {X 0,Y 639.998,Z 627.329,A -85,B 0,C 180,E1 -6567.492,E2 -6567.492} C_VEL
LIN {X 0,Y 639.963,Z 629.348,A -85,B 0,C 180,E1 -6568.747,E2 -6568.747} C_VEL
LIN {X 0,Y 639.959,Z 630.019,A -85,B 0,C 180,E1 -6570.002,E2 -6570.002} C_VEL
LIN {X 0,Y 639.963,Z 629.353,A -85,B 0,C 180,E1 -6571.256,E2 -6571.256} C_VEL
LIN {X 0,Y 639.999,Z 627.34,A -85,B 0,C 180,E1 -6572.511,E2 -6572.511} C_VEL
LIN {X 0,Y 639.956,Z 623.927,A -85,B 0,C 180,E1 -6573.767,E2 -6573.767} C_VEL
LIN {X 0,Y 639.993,Z 619.024,A -85,B 0,C 180,E1 -6575.025,E2 -6575.025} C_VEL
LIN {X 0,Y 640.096,Z 612.476,A -85,B 0,C 180,E1 -6576.284,E2 -6576.284} C_VEL
LIN {X 0,Y 640.194,Z 605.194,A -85,B 0,C 180,E1 -6577.388,E2 -6577.388} C_VEL
LIN {X 0,Y 640.371,Z 596.2,A -85,B 0,C 180,E1 -6578.493,E2 -6578.493} C_VEL
LIN {X 0,Y 640.638,Z 586.772,A -85,B 0,C 180,E1 -6579.441,E2 -6579.441} C_VEL
LIN {X 0,Y 640.96,Z 576.842,A -85,B 0,C 180,E1 -6580.273,E2 -6580.273} C_VEL
LIN {X 0,Y 641.206,Z 564.855,A -85,B 0,C 180,E1 -6581.102,E2 -6581.102} C_VEL
LIN {X 0,Y 641.555,Z 552.145,A -85,B 0,C 180,E1 -6581.814,E2 -6581.814} C_VEL
LIN {X 0,Y 641.923,Z 539.813,A -85,B 0,C 180,E1 -6582.367,E2 -6582.367} C_VEL
LIN {X 0,Y 642.195,Z 526.174,A -85,B 0,C 180,E1 -6582.841,E2 -6582.841} C_VEL
LIN {X 0,Y 642.497,Z 512.041,A -85,B 0,C 180,E1 -6583.196,E2 -6583.196} C_VEL
LIN {X 0,Y 642.736,Z 497.134,A -85,B 0,C 180,E1 -6583.432,E2 -6583.432} C_VEL
LIN {X 0,Y 643.164,Z 381.417,A -85,B 0,C 180,E1 -6584.728,E2 -6584.728} C_VEL
LIN {X 0,Y 641.143,Z 365.877,A -85,B 0,C 180,E1 -6584.959,E2 -6584.959} C_VEL
LIN {X 0,Y 641.525,Z 344.878,A -85,B 0,C 180,E1 -6587.31,E2 -6587.31} C_VEL
LIN {X 0,Y 641.959,Z 324.572,A -85,B 0,C 180,E1 -6589.605,E2 -6589.605} C_VEL
LIN {X 0,Y 642.44,Z 308.567,A -85,B 0,C 180,E1 -6591.424,E2 -6591.424} C_VEL
LIN {X 0,Y 642.969,Z 289.103,A -85,B 0,C 180,E1 -6593.663,E2 -6593.663} C_VEL
LIN {X 0,Y 640.767,Z 277.227,A -85,B 0,C 180,E1 -6595.135,E2 -6595.135} C_VEL
LIN {X 0,Y 640.723,Z 277.234,A -85,B 0,C 180,E1 -6598.041,E2 -6598.041} C_VEL
LIN {X 0,Y 640.699,Z 277.23,A -85,B 0,C 180,E1 -6600.92,E2 -6600.92} C_VEL
LIN {X 0,Y 640.719,Z 277.228,A -85,B 0,C 180,E1 -6603.136,E2 -6603.136} C_VEL
LIN {X 0,Y 640.727,Z 277.231,A -85,B 0,C 180,E1 -6606.005,E2 -6606.005} C_VEL
LIN {X 0,Y 640.717,Z 277.228,A -85,B 0,C 180,E1 -6608.547,E2 -6608.547} C_VEL
LIN {X 0,Y 640.709,Z 277.234,A -85,B 0,C 180,E1 -6611.033,E2 -6611.033} C_VEL
LIN {X 0,Y 640.699,Z 277.231,A -85,B 0,C 180,E1 -6613.818,E2 -6613.818} C_VEL
LIN {X 0,Y 640.721,Z 277.228,A -85,B 0,C 180,E1 -6616.471,E2 -6616.471} C_VEL
LIN {X 0,Y 640.713,Z 277.237,A -85,B 0,C 180,E1 -6619.009,E2 -6619.009} C_VEL
LIN {X 0,Y 640.711,Z 277.229,A -85,B 0,C 180,E1 -6621.919,E2 -6621.919} C_VEL
LIN {X 0,Y 640.765,Z 277.229,A -85,B 0,C 180,E1 -6624.594,E2 -6624.594} C_VEL
LIN {X 0,Y 640.735,Z 277.226,A -85,B 0,C 180,E1 -6627.327,E2 -6627.327} C_VEL
LIN {X 0,Y 640.744,Z 277.226,A -85,B 0,C 180,E1 -6629.811,E2 -6629.811} C_VEL
LIN {X 0,Y 640.742,Z 277.233,A -85,B 0,C 180,E1 -6632.311,E2 -6632.311} C_VEL
LIN {X 0,Y 640.761,Z 277.224,A -85,B 0,C 180,E1 -6635.138,E2 -6635.138} C_VEL
LIN {X 0,Y 640.742,Z 277.228,A -85,B 0,C 180,E1 -6637.504,E2 -6637.504} C_VEL
LIN {X 0,Y 640.787,Z 277.232,A -85,B 0,C 180,E1 -6640.192,E2 -6640.192} C_VEL
LIN {X 0,Y 640.753,Z 277.225,A -85,B 0,C 180,E1 -6642.833,E2 -6642.833} C_VEL
LIN {X 0,Y 640.746,Z 277.226,A -85,B 0,C 180,E1 -6644.79,E2 -6644.79} C_VEL
LIN {X 0,Y 640.779,Z 277.228,A -85,B 0,C 180,E1 -6647.372,E2 -6647.372} C_VEL
LIN {X 0,Y 640.795,Z 277.261,A -85,B 0,C 180,E1 -6649.339,E2 -6649.339} C_VEL
LIN {X 0,Y 642.157,Z 285.996,A -85,B 0,C 180,E1 -6650.425,E2 -6650.425} C_VEL
LIN {X 0,Y 641.981,Z 307.023,A -85,B 0,C 180,E1 -6652.949,E2 -6652.949} C_VEL
LIN {X 0,Y 641.56,Z 328.02,A -85,B 0,C 180,E1 -6655.46,E2 -6655.46} C_VEL
LIN {X 0,Y 641.424,Z 341.605,A -85,B 0,C 180,E1 -6657.105,E2 -6657.105} C_VEL
LIN {X 0,Y 643.381,Z 355.059,A -85,B 0,C 180,E1 -6657.328,E2 -6657.328} C_VEL
LIN {X 0,Y 642.48,Z 479.707,A -85,B 0,C 180,E1 -6658.829,E2 -6658.829} C_VEL
LIN {X 0,Y 642.274,Z 493.83,A -85,B 0,C 180,E1 -6659.121,E2 -6659.121} C_VEL
LIN {X 0,Y 642.032,Z 507.496,A -85,B 0,C 180,E1 -6659.531,E2 -6659.531} C_VEL
LIN {X 0,Y 641.738,Z 519.419,A -85,B 0,C 180,E1 -6660,E2 -6660} C_VEL
LIN {X 0,Y 641.427,Z 532.035,A -85,B 0,C 180,E1 -6660.626,E2 -6660.626} C_VEL
LIN {X 0,Y 641.233,Z 543.504,A -85,B 0,C 180,E1 -6661.33,E2 -6661.33} C_VEL
LIN {X 0,Y 640.959,Z 553.142,A -85,B 0,C 180,E1 -6662.035,E2 -6662.035} C_VEL
LIN {X 0,Y 640.585,Z 563.807,A -85,B 0,C 180,E1 -6662.977,E2 -6662.977} C_VEL
LIN {X 0,Y 640.389,Z 572.628,A -85,B 0,C 180,E1 -6663.92,E2 -6663.92} C_VEL
LIN {X 0,Y 640.309,Z 579.982,A -85,B 0,C 180,E1 -6664.863,E2 -6664.863} C_VEL
LIN {X 0,Y 640.131,Z 587.029,A -85,B 0,C 180,E1 -6665.967,E2 -6665.967} C_VEL
LIN {X 0,Y 640.032,Z 591.948,A -85,B 0,C 180,E1 -6666.914,E2 -6666.914} C_VEL
LIN {X 0,Y 639.921,Z 597.012,A -85,B 0,C 180,E1 -6668.181,E2 -6668.181} C_VEL
LIN {X 0,Y 639.942,Z 600.558,A -85,B 0,C 180,E1 -6669.45,E2 -6669.45} C_VEL
LIN {X 0,Y 639.859,Z 602.689,A -85,B 0,C 180,E1 -6670.725,E2 -6670.725} C_VEL
LIN {X 0,Y 639.844,Z 603.434,A -85,B 0,C 180,E1 -6672.005,E2 -6672.005} C_VEL
LIN {X 0,Y 639.9,Z 602.764,A -85,B 0,C 180,E1 -6673.289,E2 -6673.289} C_VEL
LIN {X 0,Y 639.863,Z 600.654,A -85,B 0,C 180,E1 -6674.583,E2 -6674.583} C_VEL
LIN {X 0,Y 639.96,Z 597.057,A -85,B 0,C 180,E1 -6675.88,E2 -6675.88} C_VEL
LIN {X 0,Y 640.036,Z 591.843,A -85,B 0,C 180,E1 -6677.187,E2 -6677.187} C_VEL
LIN {X 0,Y 640.135,Z 586.699,A -85,B 0,C 180,E1 -6678.171,E2 -6678.171} C_VEL
LIN {X 0,Y 640.267,Z 579.237,A -85,B 0,C 180,E1 -6679.325,E2 -6679.325} C_VEL
LIN {X 0,Y 640.462,Z 571.321,A -85,B 0,C 180,E1 -6680.318,E2 -6680.318} C_VEL
LIN {X 0,Y 640.695,Z 561.773,A -85,B 0,C 180,E1 -6681.305,E2 -6681.305} C_VEL
LIN {X 0,Y 640.966,Z 551.933,A -85,B 0,C 180,E1 -6682.149,E2 -6682.149} C_VEL
LIN {X 0,Y 641.296,Z 540.106,A -85,B 0,C 180,E1 -6682.984,E2 -6682.984} C_VEL
LIN {X 0,Y 641.599,Z 527.286,A -85,B 0,C 180,E1 -6683.719,E2 -6683.719} C_VEL
LIN {X 0,Y 641.892,Z 514.963,A -85,B 0,C 180,E1 -6684.284,E2 -6684.284} C_VEL
LIN {X 0,Y 642.197,Z 502.133,A -85,B 0,C 180,E1 -6684.743,E2 -6684.743} C_VEL
LIN {X 0,Y 642.414,Z 487.81,A -85,B 0,C 180,E1 -6685.122,E2 -6685.122} C_VEL
LIN {X 0,Y 642.557,Z 473.773,A -85,B 0,C 180,E1 -6685.363,E2 -6685.363} C_VEL
LIN {X 0,Y 643.242,Z 353.142,A -85,B 0,C 180,E1 -6686.778,E2 -6686.778} C_VEL
LIN {X 0,Y 641.329,Z 341.264,A -85,B 0,C 180,E1 -6686.969,E2 -6686.969} C_VEL
LIN {X 0,Y 641.71,Z 319.92,A -85,B 0,C 180,E1 -6689.598,E2 -6689.598} C_VEL
LIN {X 0,Y 642.082,Z 301,A -85,B 0,C 180,E1 -6691.923,E2 -6691.923} C_VEL
LIN {X 0,Y 642.24,Z 285.837,A -85,B 0,C 180,E1 -6693.795,E2 -6693.795} C_VEL
LIN {X 0,Y 642.044,Z 284.037,A -85,B 0,C 180,E1 -6694.022,E2 -6694.022} C_VEL
LIN {X 0,Y 640.969,Z 281.966,A -85,B 0,C 180,E1 -6694.318,E2 -6694.318} C_VEL
LIN {X 0,Y 637.591,Z 279.566,A -85,B 0,C 180,E1 -6694.808,E2 -6694.808} C_VEL
LIN {X 0,Y 634.933,Z 278.49,A -85,B 0,C 180,E1 -6695.226,E2 -6695.226} C_VEL
LIN {X 0,Y 633.747,Z 278.122,A -85,B 0,C 180,E1 -6695.601,E2 -6695.601} C_VEL
LIN {X 0,Y 633.696,Z 278.108,A -85,B 0,C 180,E1 -6695.691,E2 -6695.691} C_VEL
LIN {X 0,Y 633.695,Z 278.112,A -85,B 0,C 180,E1 -6698.298,E2 -6698.298} C_VEL
LIN {X 0,Y 633.658,Z 278.109,A -85,B 0,C 180,E1 -6700.707,E2 -6700.707} C_VEL
LIN {X 0,Y 633.69,Z 278.104,A -85,B 0,C 180,E1 -6703.26,E2 -6703.26} C_VEL
LIN {X 0,Y 633.681,Z 278.112,A -85,B 0,C 180,E1 -6705.929,E2 -6705.929} C_VEL
LIN {X 0,Y 633.665,Z 278.107,A -85,B 0,C 180,E1 -6708.735,E2 -6708.735} C_VEL
LIN {X 0,Y 633.645,Z 278.112,A -85,B 0,C 180,E1 -6710.942,E2 -6710.942} C_VEL
LIN {X 0,Y 633.685,Z 278.11,A -85,B 0,C 180,E1 -6713.795,E2 -6713.795} C_VEL
LIN {X 0,Y 633.672,Z 278.107,A -85,B 0,C 180,E1 -6716.447,E2 -6716.447} C_VEL
LIN {X 0,Y 633.685,Z 278.108,A -85,B 0,C 180,E1 -6718.699,E2 -6718.699} C_VEL
LIN {X 0,Y 633.697,Z 278.106,A -85,B 0,C 180,E1 -6721.62,E2 -6721.62} C_VEL
LIN {X 0,Y 633.669,Z 278.111,A -85,B 0,C 180,E1 -6724.462,E2 -6724.462} C_VEL
LIN {X 0,Y 633.72,Z 278.103,A -85,B 0,C 180,E1 -6727.24,E2 -6727.24} C_VEL
LIN {X 0,Y 633.723,Z 278.102,A -85,B 0,C 180,E1 -6729.966,E2 -6729.966} C_VEL
LIN {X 0,Y 633.724,Z 278.104,A -85,B 0,C 180,E1 -6732.636,E2 -6732.636} C_VEL
LIN {X 0,Y 633.739,Z 278.098,A -85,B 0,C 180,E1 -6735.272,E2 -6735.272} C_VEL
LIN {X 0,Y 633.735,Z 278.103,A -85,B 0,C 180,E1 -6737.876,E2 -6737.876} C_VEL
LIN {X 0,Y 633.785,Z 278.096,A -85,B 0,C 180,E1 -6740.456,E2 -6740.456} C_VEL
LIN {X 0,Y 633.785,Z 278.095,A -85,B 0,C 180,E1 -6743.016,E2 -6743.016} C_VEL
LIN {X 0,Y 633.864,Z 278.167,A -85,B 0,C 180,E1 -6743.946,E2 -6743.946} C_VEL
LIN {X 0,Y 634.498,Z 283.951,A -85,B 0,C 180,E1 -6744.932,E2 -6744.932} C_VEL
LIN {X 0,Y 634.255,Z 296.278,A -85,B 0,C 180,E1 -6746.972,E2 -6746.972} C_VEL
LIN {X 0,Y 636.613,Z 307.905,A -85,B 0,C 180,E1 -6747.161,E2 -6747.161} C_VEL
LIN {X 0,Y 635.876,Z 431.815,A -85,B 0,C 180,E1 -6748.578,E2 -6748.578} C_VEL
LIN {X 0,Y 635.731,Z 446.093,A -85,B 0,C 180,E1 -6748.874,E2 -6748.874} C_VEL
LIN {X 0,Y 635.496,Z 459.824,A -85,B 0,C 180,E1 -6749.288,E2 -6749.288} C_VEL
LIN {X 0,Y 635.213,Z 471.766,A -85,B 0,C 180,E1 -6749.762,E2 -6749.762} C_VEL
LIN {X 0,Y 634.902,Z 484.347,A -85,B 0,C 180,E1 -6750.394,E2 -6750.394} C_VEL
LIN {X 0,Y 634.532,Z 495.832,A -85,B 0,C 180,E1 -6751.105,E2 -6751.105} C_VEL
LIN {X 0,Y 634.241,Z 506.353,A -85,B 0,C 180,E1 -6751.897,E2 -6751.897} C_VEL
LIN {X 0,Y 633.844,Z 516.824,A -85,B 0,C 180,E1 -6752.849,E2 -6752.849} C_VEL
LIN {X 0,Y 633.621,Z 525.465,A -85,B 0,C 180,E1 -6753.801,E2 -6753.801} C_VEL
LIN {X 0,Y 633.34,Z 533.79,A -85,B 0,C 180,E1 -6754.915,E2 -6754.915} C_VEL
LIN {X 0,Y 633.213,Z 540.496,A -85,B 0,C 180,E1 -6756.03,E2 -6756.03} C_VEL
LIN {X 0,Y 633.102,Z 545.125,A -85,B 0,C 180,E1 -6756.989,E2 -6756.989} C_VEL
LIN {X 0,Y 632.944,Z 549.942,A -85,B 0,C 180,E1 -6758.27,E2 -6758.27} C_VEL
LIN {X 0,Y 632.938,Z 553.274,A -85,B 0,C 180,E1 -6759.554,E2 -6759.554} C_VEL
LIN {X 0,Y 632.885,Z 555.217,A -85,B 0,C 180,E1 -6760.843,E2 -6760.843} C_VEL
LIN {X 0,Y 632.864,Z 555.797,A -85,B 0,C 180,E1 -6762.138,E2 -6762.138} C_VEL
LIN {X 0,Y 632.909,Z 555.017,A -85,B 0,C 180,E1 -6763.437,E2 -6763.437} C_VEL
LIN {X 0,Y 632.894,Z 552.852,A -85,B 0,C 180,E1 -6764.745,E2 -6764.745} C_VEL
LIN {X 0,Y 633.042,Z 549.22,A -85,B 0,C 180,E1 -6766.057,E2 -6766.057} C_VEL
LIN {X 0,Y 633.129,Z 543.992,A -85,B 0,C 180,E1 -6767.378,E2 -6767.378} C_VEL
LIN {X 0,Y 633.289,Z 538.853,A -85,B 0,C 180,E1 -6768.372,E2 -6768.372} C_VEL
LIN {X 0,Y 633.51,Z 531.429,A -85,B 0,C 180,E1 -6769.536,E2 -6769.536} C_VEL
LIN {X 0,Y 633.709,Z 523.525,A -85,B 0,C 180,E1 -6770.543,E2 -6770.543} C_VEL
LIN {X 0,Y 634.065,Z 514.208,A -85,B 0,C 180,E1 -6771.522,E2 -6771.522} C_VEL
LIN {X 0,Y 634.347,Z 503.161,A -85,B 0,C 180,E1 -6772.476,E2 -6772.476} C_VEL
LIN {X 0,Y 634.731,Z 492.488,A -85,B 0,C 180,E1 -6773.233,E2 -6773.233} C_VEL
LIN {X 0,Y 635.022,Z 480.064,A -85,B 0,C 180,E1 -6773.956,E2 -6773.956} C_VEL
LIN {X 0,Y 635.424,Z 466.239,A -85,B 0,C 180,E1 -6774.588,E2 -6774.588} C_VEL
LIN {X 0,Y 635.706,Z 452.941,A -85,B 0,C 180,E1 -6775.053,E2 -6775.053} C_VEL
LIN {X 0,Y 635.89,Z 439.571,A -85,B 0,C 180,E1 -6775.394,E2 -6775.394} C_VEL
LIN {X 0,Y 635.965,Z 425.068,A -85,B 0,C 180,E1 -6775.633,E2 -6775.633} C_VEL
LIN {X 0,Y 636.517,Z 306.839,A -85,B 0,C 180,E1 -6776.98,E2 -6776.98} C_VEL
LIN {X 0,Y 634.382,Z 296.436,A -85,B 0,C 180,E1 -6777.171,E2 -6777.171} C_VEL
LIN {X 0,Y 634.596,Z 283.679,A -85,B 0,C 180,E1 -6779.311,E2 -6779.311} C_VEL
LIN {X 0,Y 633.682,Z 278.113,A -85,B 0,C 180,E1 -6780.315,E2 -6780.315} C_VEL
LIN {X 0,Y 633.666,Z 278.109,A -85,B 0,C 180,E1 -6782.85,E2 -6782.85} C_VEL
LIN {X 0,Y 633.667,Z 278.107,A -85,B 0,C 180,E1 -6785.117,E2 -6785.117} C_VEL
LIN {X 0,Y 633.646,Z 278.109,A -85,B 0,C 180,E1 -6787.441,E2 -6787.441} C_VEL
LIN {X 0,Y 633.653,Z 278.114,A -85,B 0,C 180,E1 -6790.294,E2 -6790.294} C_VEL
LIN {X 0,Y 633.67,Z 278.107,A -85,B 0,C 180,E1 -6793.259,E2 -6793.259} C_VEL
LIN {X 0,Y 633.66,Z 278.111,A -85,B 0,C 180,E1 -6795.928,E2 -6795.928} C_VEL
LIN {X 0,Y 633.688,Z 278.103,A -85,B 0,C 180,E1 -6798.729,E2 -6798.729} C_VEL
LIN {X 0,Y 633.668,Z 278.113,A -85,B 0,C 180,E1 -6801.7,E2 -6801.7} C_VEL
LIN {X 0,Y 633.682,Z 278.1,A -85,B 0,C 180,E1 -6804.138,E2 -6804.138} C_VEL
LIN {X 0,Y 633.651,Z 278.108,A -85,B 0,C 180,E1 -6806.447,E2 -6806.447} C_VEL
LIN {X 0,Y 633.668,Z 278.103,A -85,B 0,C 180,E1 -6808.699,E2 -6808.699} C_VEL
LIN {X 0,Y 633.716,Z 278.099,A -85,B 0,C 180,E1 -6810.9,E2 -6810.9} C_VEL
LIN {X 0,Y 633.65,Z 278.113,A -85,B 0,C 180,E1 -6813.552,E2 -6813.552} C_VEL
LIN {X 0,Y 633.697,Z 278.104,A -85,B 0,C 180,E1 -6815.86,E2 -6815.86} C_VEL
LIN {X 0,Y 633.692,Z 278.102,A -85,B 0,C 180,E1 -6818.607,E2 -6818.607} C_VEL
LIN {X 0,Y 633.677,Z 278.108,A -85,B 0,C 180,E1 -6821.303,E2 -6821.303} C_VEL
LIN {X 0,Y 633.723,Z 278.099,A -85,B 0,C 180,E1 -6824.061,E2 -6824.061} C_VEL
LIN {X 0,Y 633.758,Z 278.09,A -85,B 0,C 180,E1 -6826.579,E2 -6826.579} C_VEL
LIN {X 0,Y 633.712,Z 278.102,A -85,B 0,C 180,E1 -6829.634,E2 -6829.634} C_VEL
LIN {X 0,Y 633.785,Z 278.088,A -85,B 0,C 180,E1 -6832.379,E2 -6832.379} C_VEL
LIN {X 0,Y 633.807,Z 278.093,A -85,B 0,C 180,E1 -6834.928,E2 -6834.928} C_VEL
LIN {X 0,Y 633.808,Z 278.086,A -85,B 0,C 180,E1 -6838.1,E2 -6838.1} C_VEL
LIN {X 0,Y 633.858,Z 278.08,A -85,B 0,C 180,E1 -6840,E2 -6840} C_VEL
LIN {X 0,Y 633.84,Z 278.078,A -85,B 0,C 180,E1 -6841.9,E2 -6841.9} C_VEL
LIN {X 0,Y 633.822,Z 278.094,A -85,B 0,C 180,E1 -6845.072,E2 -6845.072} C_VEL
LIN {X 0,Y 633.786,Z 278.086,A -85,B 0,C 180,E1 -6847.621,E2 -6847.621} C_VEL
LIN {X 0,Y 633.777,Z 278.093,A -85,B 0,C 180,E1 -6850.398,E2 -6850.398} C_VEL
LIN {X 0,Y 633.755,Z 278.093,A -85,B 0,C 180,E1 -6853.454,E2 -6853.454} C_VEL
LIN {X 0,Y 633.732,Z 278.096,A -85,B 0,C 180,E1 -6856.041,E2 -6856.041} C_VEL
LIN {X 0,Y 633.69,Z 278.107,A -85,B 0,C 180,E1 -6858.696,E2 -6858.696} C_VEL
LIN {X 0,Y 633.695,Z 278.099,A -85,B 0,C 180,E1 -6861.393,E2 -6861.393} C_VEL
LIN {X 0,Y 633.699,Z 278.103,A -85,B 0,C 180,E1 -6864.14,E2 -6864.14} C_VEL
LIN {X 0,Y 633.652,Z 278.11,A -85,B 0,C 180,E1 -6866.95,E2 -6866.95} C_VEL
LIN {X 0,Y 633.698,Z 278.102,A -85,B 0,C 180,E1 -6869.171,E2 -6869.171} C_VEL
LIN {X 0,Y 633.691,Z 278.105,A -85,B 0,C 180,E1 -6872.044,E2 -6872.044} C_VEL
LIN {X 0,Y 633.711,Z 278.09,A -85,B 0,C 180,E1 -6875.126,E2 -6875.126} C_VEL
LIN {X 0,Y 633.706,Z 278.097,A -85,B 0,C 180,E1 -6877.44,E2 -6877.44} C_VEL
LIN {X 0,Y 633.686,Z 278.11,A -85,B 0,C 180,E1 -6880.302,E2 -6880.302} C_VEL
LIN {X 0,Y 633.69,Z 278.102,A -85,B 0,C 180,E1 -6883.157,E2 -6883.157} C_VEL
LIN {X 0,Y 633.675,Z 278.108,A -85,B 0,C 180,E1 -6885.93,E2 -6885.93} C_VEL
LIN {X 0,Y 633.69,Z 278.108,A -85,B 0,C 180,E1 -6888.458,E2 -6888.458} C_VEL
LIN {X 0,Y 633.676,Z 278.104,A -85,B 0,C 180,E1 -6890.948,E2 -6890.948} C_VEL
LIN {X 0,Y 633.719,Z 278.103,A -85,B 0,C 180,E1 -6893.791,E2 -6893.791} C_VEL
LIN {X 0,Y 633.669,Z 278.112,A -85,B 0,C 180,E1 -6896.451,E2 -6896.451} C_VEL
LIN {X 0,Y 633.687,Z 278.108,A -85,B 0,C 180,E1 -6898.703,E2 -6898.703} C_VEL
LIN {X 0,Y 633.729,Z 278.1,A -85,B 0,C 180,E1 -6900.903,E2 -6900.903} C_VEL
LIN {X 0,Y 633.671,Z 278.112,A -85,B 0,C 180,E1 -6903.554,E2 -6903.554} C_VEL
LIN {X 0,Y 633.716,Z 278.233,A -85,B 0,C 180,E1 -6904.6,E2 -6904.6} C_VEL
LIN {X 0,Y 636.163,Z 290.524,A -85,B 0,C 180,E1 -6906.187,E2 -6906.187} C_VEL
LIN {X 0,Y 635.505,Z 313.017,A -85,B 0,C 180,E1 -6908.842,E2 -6908.842} C_VEL
LIN {X 0,Y 634.71,Z 340.317,A -85,B 0,C 180,E1 -6912.003,E2 -6912.003} C_VEL
LIN {X 0,Y 634.111,Z 365.292,A -85,B 0,C 180,E1 -6914.854,E2 -6914.854} C_VEL
LIN {X 0,Y 636.441,Z 384.069,A -85,B 0,C 180,E1 -6915.135,E2 -6915.135} C_VEL
LIN {X 0,Y 635.81,Z 503.434,A -85,B 0,C 180,E1 -6916.504,E2 -6916.504} C_VEL
LIN {X 0,Y 635.507,Z 517.334,A -85,B 0,C 180,E1 -6916.781,E2 -6916.781} C_VEL
LIN {X 0,Y 635.207,Z 530.959,A -85,B 0,C 180,E1 -6917.18,E2 -6917.18} C_VEL
LIN {X 0,Y 634.881,Z 543.347,A -85,B 0,C 180,E1 -6917.659,E2 -6917.659} C_VEL
LIN {X 0,Y 634.428,Z 556.321,A -85,B 0,C 180,E1 -6918.297,E2 -6918.297} C_VEL
LIN {X 0,Y 634.147,Z 568.109,A -85,B 0,C 180,E1 -6919.018,E2 -6919.018} C_VEL
LIN {X 0,Y 633.849,Z 578.911,A -85,B 0,C 180,E1 -6919.818,E2 -6919.818} C_VEL
LIN {X 0,Y 633.515,Z 589.62,A -85,B 0,C 180,E1 -6920.776,E2 -6920.776} C_VEL
LIN {X 0,Y 633.233,Z 598.476,A -85,B 0,C 180,E1 -6921.734,E2 -6921.734} C_VEL
LIN {X 0,Y 633.092,Z 605.859,A -85,B 0,C 180,E1 -6922.692,E2 -6922.692} C_VEL
LIN {X 0,Y 633.003,Z 612.02,A -85,B 0,C 180,E1 -6923.649,E2 -6923.649} C_VEL
LIN {X 0,Y 632.924,Z 618.576,A -85,B 0,C 180,E1 -6924.922,E2 -6924.922} C_VEL
LIN {X 0,Y 632.885,Z 623.494,A -85,B 0,C 180,E1 -6926.194,E2 -6926.194} C_VEL
LIN {X 0,Y 632.901,Z 626.913,A -85,B 0,C 180,E1 -6927.464,E2 -6927.464} C_VEL
LIN {X 0,Y 632.882,Z 628.934,A -85,B 0,C 180,E1 -6928.733,E2 -6928.733} C_VEL
LIN {X 0,Y 632.871,Z 629.605,A -85,B 0,C 180,E1 -6930.002,E2 -6930.002} C_VEL
LIN {X 0,Y 632.882,Z 628.941,A -85,B 0,C 180,E1 -6931.27,E2 -6931.27} C_VEL
LIN {X 0,Y 632.902,Z 626.927,A -85,B 0,C 180,E1 -6932.539,E2 -6932.539} C_VEL
LIN {X 0,Y 632.886,Z 623.516,A -85,B 0,C 180,E1 -6933.809,E2 -6933.809} C_VEL
LIN {X 0,Y 632.927,Z 618.611,A -85,B 0,C 180,E1 -6935.081,E2 -6935.081} C_VEL
LIN {X 0,Y 633.006,Z 612.059,A -85,B 0,C 180,E1 -6936.354,E2 -6936.354} C_VEL
LIN {X 0,Y 633.113,Z 604.772,A -85,B 0,C 180,E1 -6937.471,E2 -6937.471} C_VEL
LIN {X 0,Y 633.313,Z 595.773,A -85,B 0,C 180,E1 -6938.588,E2 -6938.588} C_VEL
LIN {X 0,Y 633.574,Z 586.335,A -85,B 0,C 180,E1 -6939.547,E2 -6939.547} C_VEL
LIN {X 0,Y 633.915,Z 575.547,A -85,B 0,C 180,E1 -6940.452,E2 -6940.452} C_VEL
LIN {X 0,Y 634.199,Z 564.4,A -85,B 0,C 180,E1 -6941.226,E2 -6941.226} C_VEL
LIN {X 0,Y 634.567,Z 551.667,A -85,B 0,C 180,E1 -6941.946,E2 -6941.946} C_VEL
LIN {X 0,Y 634.96,Z 539.306,A -85,B 0,C 180,E1 -6942.504,E2 -6942.504} C_VEL
LIN {X 0,Y 635.259,Z 525.623,A -85,B 0,C 180,E1 -6942.984,E2 -6942.984} C_VEL
LIN {X 0,Y 635.574,Z 511.418,A -85,B 0,C 180,E1 -6943.342,E2 -6943.342} C_VEL
LIN {X 0,Y 635.811,Z 497.89,A -85,B 0,C 180,E1 -6943.56,E2 -6943.56} C_VEL
LIN {X 0,Y 636.25,Z 382.117,A -85,B 0,C 180,E1 -6944.872,E2 -6944.872} C_VEL
LIN {X 0,Y 634.104,Z 365.398,A -85,B 0,C 180,E1 -6945.129,E2 -6945.129} C_VEL
LIN {X 0,Y 634.572,Z 342.972,A -85,B 0,C 180,E1 -6947.672,E2 -6947.672} C_VEL
LIN {X 0,Y 635.053,Z 322.624,A -85,B 0,C 180,E1 -6949.995,E2 -6949.995} C_VEL
LIN {X 0,Y 635.732,Z 301.652,A -85,B 0,C 180,E1 -6952.415,E2 -6952.415} C_VEL
LIN {X 0,Y 635.986,Z 289.872,A -85,B 0,C 180,E1 -6953.789,E2 -6953.789} C_VEL
LIN {X 0,Y 633.709,Z 278.107,A -85,B 0,C 180,E1 -6955.287,E2 -6955.287} C_VEL
LIN {X 0,Y 633.699,Z 278.11,A -85,B 0,C 180,E1 -6957.839,E2 -6957.839} C_VEL
LIN {X 0,Y 633.649,Z 278.111,A -85,B 0,C 180,E1 -6960.433,E2 -6960.433} C_VEL
LIN {X 0,Y 633.679,Z 278.104,A -85,B 0,C 180,E1 -6962.852,E2 -6962.852} C_VEL
LIN {X 0,Y 633.687,Z 278.107,A -85,B 0,C 180,E1 -6965.119,E2 -6965.119} C_VEL
LIN {X 0,Y 633.664,Z 278.115,A -85,B 0,C 180,E1 -6967.444,E2 -6967.444} C_VEL
LIN {X 0,Y 633.671,Z 278.106,A -85,B 0,C 180,E1 -6970.296,E2 -6970.296} C_VEL
LIN {X 0,Y 633.68,Z 278.113,A -85,B 0,C 180,E1 -6973.262,E2 -6973.262} C_VEL
LIN {X 0,Y 633.678,Z 278.105,A -85,B 0,C 180,E1 -6975.931,E2 -6975.931} C_VEL
LIN {X 0,Y 633.666,Z 278.111,A -85,B 0,C 180,E1 -6978.736,E2 -6978.736} C_VEL
LIN {X 0,Y 633.648,Z 278.117,A -85,B 0,C 180,E1 -6980.943,E2 -6980.943} C_VEL
LIN {X 0,Y 633.71,Z 278.101,A -85,B 0,C 180,E1 -6983.793,E2 -6983.793} C_VEL
LIN {X 0,Y 633.676,Z 278.111,A -85,B 0,C 180,E1 -6986.449,E2 -6986.449} C_VEL
LIN {X 0,Y 633.688,Z 278.111,A -85,B 0,C 180,E1 -6988.7,E2 -6988.7} C_VEL
LIN {X 0,Y 633.699,Z 278.102,A -85,B 0,C 180,E1 -6991.622,E2 -6991.622} C_VEL
LIN {X 0,Y 633.671,Z 278.114,A -85,B 0,C 180,E1 -6994.463,E2 -6994.463} C_VEL
LIN {X 0,Y 633.722,Z 278.102,A -85,B 0,C 180,E1 -6997.241,E2 -6997.241} C_VEL
LIN {X 0,Y 633.725,Z 278.112,A -85,B 0,C 180,E1 -6999.968,E2 -6999.968} C_VEL
LIN {X 0,Y 633.71,Z 278.104,A -85,B 0,C 180,E1 -7002.636,E2 -7002.636} C_VEL
LIN {X 0,Y 633.732,Z 278.101,A -85,B 0,C 180,E1 -7004.617,E2 -7004.617} C_VEL
LIN {X 0,Y 633.759,Z 278.101,A -85,B 0,C 180,E1 -7007.23,E2 -7007.23} C_VEL
LIN {X 0,Y 633.77,Z 278.204,A -85,B 0,C 180,E1 -7009.211,E2 -7009.211} C_VEL
LIN {X 0,Y 635.21,Z 287.037,A -85,B 0,C 180,E1 -7010.319,E2 -7010.319} C_VEL
LIN {X 0,Y 635.048,Z 308.263,A -85,B 0,C 180,E1 -7012.872,E2 -7012.872} C_VEL
LIN {X 0,Y 634.577,Z 329.307,A -85,B 0,C 180,E1 -7015.41,E2 -7015.41} C_VEL
LIN {X 0,Y 634.481,Z 341.82,A -85,B 0,C 180,E1 -7016.935,E2 -7016.935} C_VEL
LIN {X 0,Y 636.523,Z 355.273,A -85,B 0,C 180,E1 -7017.162,E2 -7017.162} C_VEL
LIN {X 0,Y 635.564,Z 479.062,A -85,B 0,C 180,E1 -7018.678,E2 -7018.678} C_VEL
LIN {X 0,Y 635.387,Z 493.418,A -85,B 0,C 180,E1 -7018.974,E2 -7018.974} C_VEL
LIN {X 0,Y 635.068,Z 507.842,A -85,B 0,C 180,E1 -7019.408,E2 -7019.408} C_VEL
LIN {X 0,Y 634.737,Z 520.575,A -85,B 0,C 180,E1 -7019.921,E2 -7019.921} C_VEL
LIN {X 0,Y 634.421,Z 532.969,A -85,B 0,C 180,E1 -7020.553,E2 -7020.553} C_VEL
LIN {X 0,Y 634.172,Z 545.429,A -85,B 0,C 180,E1 -7021.345,E2 -7021.345} C_VEL
LIN {X 0,Y 633.778,Z 556.677,A -85,B 0,C 180,E1 -7022.217,E2 -7022.217} C_VEL
LIN {X 0,Y 633.551,Z 566.77,A -85,B 0,C 180,E1 -7023.169,E2 -7023.169} C_VEL
LIN {X 0,Y 633.215,Z 575.16,A -85,B 0,C 180,E1 -7024.123,E2 -7024.123} C_VEL
LIN {X 0,Y 633.137,Z 582.111,A -85,B 0,C 180,E1 -7025.078,E2 -7025.078} C_VEL
LIN {X 0,Y 633.036,Z 587.896,A -85,B 0,C 180,E1 -7026.034,E2 -7026.034} C_VEL
LIN {X 0,Y 632.932,Z 594.078,A -85,B 0,C 180,E1 -7027.312,E2 -7027.312} C_VEL
LIN {X 0,Y 632.836,Z 597.594,A -85,B 0,C 180,E1 -7028.273,E2 -7028.273} C_VEL
LIN {X 0,Y 632.857,Z 601.005,A -85,B 0,C 180,E1 -7029.556,E2 -7029.556} C_VEL
LIN {X 0,Y 632.761,Z 602.997,A -85,B 0,C 180,E1 -7030.847,E2 -7030.847} C_VEL
LIN {X 0,Y 632.768,Z 603.565,A -85,B 0,C 180,E1 -7032.141,E2 -7032.141} C_VEL
LIN {X 0,Y 632.814,Z 602.731,A -85,B 0,C 180,E1 -7033.441,E2 -7033.441} C_VEL
LIN {X 0,Y 632.804,Z 600.47,A -85,B 0,C 180,E1 -7034.749,E2 -7034.749} C_VEL
LIN {X 0,Y 632.905,Z 596.714,A -85,B 0,C 180,E1 -7036.062,E2 -7036.062} C_VEL
LIN {X 0,Y 632.937,Z 592.789,A -85,B 0,C 180,E1 -7037.053,E2 -7037.053} C_VEL
LIN {X 0,Y 633.041,Z 587.856,A -85,B 0,C 180,E1 -7038.048,E2 -7038.048} C_VEL
LIN {X 0,Y 633.187,Z 580.625,A -85,B 0,C 180,E1 -7039.214,E2 -7039.214} C_VEL
LIN {X 0,Y 633.38,Z 572.964,A -85,B 0,C 180,E1 -7040.218,E2 -7040.218} C_VEL
LIN {X 0,Y 633.611,Z 563.645,A -85,B 0,C 180,E1 -7041.226,E2 -7041.226} C_VEL
LIN {X 0,Y 633.952,Z 553.279,A -85,B 0,C 180,E1 -7042.151,E2 -7042.151} C_VEL
LIN {X 0,Y 634.281,Z 541.74,A -85,B 0,C 180,E1 -7042.995,E2 -7042.995} C_VEL
LIN {X 0,Y 634.572,Z 529.729,A -85,B 0,C 180,E1 -7043.712,E2 -7043.712} C_VEL
LIN {X 0,Y 634.851,Z 517.341,A -85,B 0,C 180,E1 -7044.31,E2 -7044.31} C_VEL
LIN {X 0,Y 635.186,Z 503.978,A -85,B 0,C 180,E1 -7044.814,E2 -7044.814} C_VEL
LIN {X 0,Y 635.448,Z 490.083,A -85,B 0,C 180,E1 -7045.203,E2 -7045.203} C_VEL
LIN {X 0,Y 635.618,Z 475.517,A -85,B 0,C 180,E1 -7045.475,E2 -7045.475} C_VEL
LIN {X 0,Y 636.363,Z 353.92,A -85,B 0,C 180,E1 -7046.928,E2 -7046.928} C_VEL
LIN {X 0,Y 634.328,Z 341.271,A -85,B 0,C 180,E1 -7047.147,E2 -7047.147} C_VEL
LIN {X 0,Y 634.729,Z 320.024,A -85,B 0,C 180,E1 -7049.775,E2 -7049.775} C_VEL
LIN {X 0,Y 635.098,Z 300.799,A -85,B 0,C 180,E1 -7052.151,E2 -7052.151} C_VEL
LIN {X 0,Y 635.286,Z 287.224,A -85,B 0,C 180,E1 -7053.834,E2 -7053.834} C_VEL
LIN {X 0,Y 633.733,Z 278.104,A -85,B 0,C 180,E1 -7055.033,E2 -7055.033} C_VEL
LIN {X 0,Y 633.696,Z 278.108,A -85,B 0,C 180,E1 -7055.691,E2 -7055.691} C_VEL
LIN {X 0,Y 633.038,Z 278.193,A -85,B 0,C 180,E1 -7056.222,E2 -7056.222} C_VEL
LIN {X 0,Y 630.161,Z 278.549,A -85,B 0,C 180,E1 -7057.083,E2 -7057.083} C_VEL
LIN {X 0,Y 627.738,Z 278.849,A -85,B 0,C 180,E1 -7057.776,E2 -7057.776} C_VEL
LIN {X 0,Y 626.721,Z 278.98,A -85,B 0,C 180,E1 -7058.31,E2 -7058.31} C_VEL
LIN {X 0,Y 626.651,Z 278.985,A -85,B 0,C 180,E1 -7058.491,E2 -7058.491} C_VEL
LIN {X 0,Y 626.629,Z 278.985,A -85,B 0,C 180,E1 -7061.501,E2 -7061.501} C_VEL
LIN {X 0,Y 626.642,Z 278.987,A -85,B 0,C 180,E1 -7063.87,E2 -7063.87} C_VEL
LIN {X 0,Y 626.642,Z 278.983,A -85,B 0,C 180,E1 -7066.598,E2 -7066.598} C_VEL
LIN {X 0,Y 626.618,Z 278.99,A -85,B 0,C 180,E1 -7069.583,E2 -7069.583} C_VEL
LIN {X 0,Y 626.626,Z 278.987,A -85,B 0,C 180,E1 -7072.062,E2 -7072.062} C_VEL
LIN {X 0,Y 626.628,Z 278.986,A -85,B 0,C 180,E1 -7074.686,E2 -7074.686} C_VEL
LIN {X 0,Y 626.649,Z 278.987,A -85,B 0,C 180,E1 -7077.551,E2 -7077.551} C_VEL
LIN {X 0,Y 626.617,Z 278.987,A -85,B 0,C 180,E1 -7079.799,E2 -7079.799} C_VEL
LIN {X 0,Y 626.661,Z 278.981,A -85,B 0,C 180,E1 -7082.008,E2 -7082.008} C_VEL
LIN {X 0,Y 626.662,Z 278.984,A -85,B 0,C 180,E1 -7084.873,E2 -7084.873} C_VEL
LIN {X 0,Y 626.666,Z 278.98,A -85,B 0,C 180,E1 -7087.663,E2 -7087.663} C_VEL
LIN {X 0,Y 626.663,Z 278.987,A -85,B 0,C 180,E1 -7090.407,E2 -7090.407} C_VEL
LIN {X 0,Y 626.681,Z 278.983,A -85,B 0,C 180,E1 -7092.434,E2 -7092.434} C_VEL
LIN {X 0,Y 626.706,Z 278.974,A -85,B 0,C 180,E1 -7095.103,E2 -7095.103} C_VEL
LIN {X 0,Y 626.69,Z 278.979,A -85,B 0,C 180,E1 -7097.738,E2 -7097.738} C_VEL
LIN {X 0,Y 626.736,Z 278.976,A -85,B 0,C 180,E1 -7100.348,E2 -7100.348} C_VEL
LIN {X 0,Y 626.761,Z 278.97,A -85,B 0,C 180,E1 -7102.937,E2 -7102.937} C_VEL
LIN {X 0,Y 626.841,Z 279.172,A -85,B 0,C 180,E1 -7103.866,E2 -7103.866} C_VEL
LIN {X 0,Y 627.506,Z 285.028,A -85,B 0,C 180,E1 -7104.875,E2 -7104.875} C_VEL
LIN {X 0,Y 627.302,Z 296.589,A -85,B 0,C 180,E1 -7106.798,E2 -7106.798} C_VEL
LIN {X 0,Y 629.758,Z 308.769,A -85,B 0,C 180,E1 -7107.01,E2 -7107.01} C_VEL
LIN {X 0,Y 628.972,Z 431.403,A -85,B 0,C 180,E1 -7108.423,E2 -7108.423} C_VEL
LIN {X 0,Y 628.837,Z 445.971,A -85,B 0,C 180,E1 -7108.722,E2 -7108.722} C_VEL
LIN {X 0,Y 628.608,Z 459.281,A -85,B 0,C 180,E1 -7109.121,E2 -7109.121} C_VEL
LIN {X 0,Y 628.286,Z 471.442,A -85,B 0,C 180,E1 -7109.599,E2 -7109.599} C_VEL
LIN {X 0,Y 627.981,Z 484.162,A -85,B 0,C 180,E1 -7110.238,E2 -7110.238} C_VEL
LIN {X 0,Y 627.536,Z 496.919,A -85,B 0,C 180,E1 -7111.038,E2 -7111.038} C_VEL
LIN {X 0,Y 627.21,Z 508.289,A -85,B 0,C 180,E1 -7111.918,E2 -7111.918} C_VEL
LIN {X 0,Y 626.8,Z 518.515,A -85,B 0,C 180,E1 -7112.881,E2 -7112.881} C_VEL
LIN {X 0,Y 626.547,Z 526.952,A -85,B 0,C 180,E1 -7113.844,E2 -7113.844} C_VEL
LIN {X 0,Y 626.289,Z 535.056,A -85,B 0,C 180,E1 -7114.971,E2 -7114.971} C_VEL
LIN {X 0,Y 626.139,Z 541.585,A -85,B 0,C 180,E1 -7116.099,E2 -7116.099} C_VEL
LIN {X 0,Y 625.985,Z 547.399,A -85,B 0,C 180,E1 -7117.392,E2 -7117.392} C_VEL
LIN {X 0,Y 625.862,Z 550.774,A -85,B 0,C 180,E1 -7118.364,E2 -7118.364} C_VEL
LIN {X 0,Y 625.875,Z 553.933,A -85,B 0,C 180,E1 -7119.662,E2 -7119.662} C_VEL
LIN {X 0,Y 625.795,Z 555.73,A -85,B 0,C 180,E1 -7120.967,E2 -7120.967} C_VEL
LIN {X 0,Y 625.793,Z 556.177,A -85,B 0,C 180,E1 -7122.277,E2 -7122.277} C_VEL
LIN {X 0,Y 625.816,Z 555.268,A -85,B 0,C 180,E1 -7123.592,E2 -7123.592} C_VEL
LIN {X 0,Y 625.847,Z 552.969,A -85,B 0,C 180,E1 -7124.915,E2 -7124.915} C_VEL
LIN {X 0,Y 625.999,Z 549.195,A -85,B 0,C 180,E1 -7126.242,E2 -7126.242} C_VEL
LIN {X 0,Y 626.044,Z 545.273,A -85,B 0,C 180,E1 -7127.245,E2 -7127.245} C_VEL
LIN {X 0,Y 626.215,Z 540.374,A -85,B 0,C 180,E1 -7128.25,E2 -7128.25} C_VEL
LIN {X 0,Y 626.43,Z 533.208,A -85,B 0,C 180,E1 -7129.428,E2 -7129.428} C_VEL
LIN {X 0,Y 626.679,Z 525.622,A -85,B 0,C 180,E1 -7130.441,E2 -7130.441} C_VEL
LIN {X 0,Y 626.993,Z 516.399,A -85,B 0,C 180,E1 -7131.459,E2 -7131.459} C_VEL
LIN {X 0,Y 627.375,Z 506.12,A -85,B 0,C 180,E1 -7132.393,E2 -7132.393} C_VEL
LIN {X 0,Y 627.725,Z 494.719,A -85,B 0,C 180,E1 -7133.247,E2 -7133.247} C_VEL
LIN {X 0,Y 628.103,Z 483.207,A -85,B 0,C 180,E1 -7133.951,E2 -7133.951} C_VEL
LIN {X 0,Y 628.412,Z 471.568,A -85,B 0,C 180,E1 -7134.53,E2 -7134.53} C_VEL
LIN {X 0,Y 628.747,Z 458.5,A -85,B 0,C 180,E1 -7135.043,E2 -7135.043} C_VEL
LIN {X 0,Y 628.938,Z 444.627,A -85,B 0,C 180,E1 -7135.449,E2 -7135.449} C_VEL
LIN {X 0,Y 629.103,Z 431.101,A -85,B 0,C 180,E1 -7135.716,E2 -7135.716} C_VEL
LIN {X 0,Y 629.737,Z 307.941,A -85,B 0,C 180,E1 -7137.149,E2 -7137.149} C_VEL
LIN {X 0,Y 627.439,Z 296.903,A -85,B 0,C 180,E1 -7137.349,E2 -7137.349} C_VEL
LIN {X 0,Y 627.611,Z 284.711,A -85,B 0,C 180,E1 -7139.408,E2 -7139.408} C_VEL
LIN {X 0,Y 626.635,Z 278.991,A -85,B 0,C 180,E1 -7140.441,E2 -7140.441} C_VEL
LIN {X 0,Y 626.618,Z 278.986,A -85,B 0,C 180,E1 -7143.209,E2 -7143.209} C_VEL
LIN {X 0,Y 626.629,Z 278.985,A -85,B 0,C 180,E1 -7145.536,E2 -7145.536} C_VEL
LIN {X 0,Y 626.632,Z 278.985,A -85,B 0,C 180,E1 -7148.514,E2 -7148.514} C_VEL
LIN {X 0,Y 626.613,Z 278.986,A -85,B 0,C 180,E1 -7151.501,E2 -7151.501} C_VEL
LIN {X 0,Y 626.619,Z 278.993,A -85,B 0,C 180,E1 -7153.869,E2 -7153.869} C_VEL
LIN {X 0,Y 626.628,Z 278.984,A -85,B 0,C 180,E1 -7156.596,E2 -7156.596} C_VEL
LIN {X 0,Y 626.642,Z 278.981,A -85,B 0,C 180,E1 -7158.739,E2 -7158.739} C_VEL
LIN {X 0,Y 626.627,Z 278.986,A -85,B 0,C 180,E1 -7161.483,E2 -7161.483} C_VEL
LIN {X 0,Y 626.662,Z 278.979,A -85,B 0,C 180,E1 -7163.672,E2 -7163.672} C_VEL
LIN {X 0,Y 626.632,Z 278.988,A -85,B 0,C 180,E1 -7166.021,E2 -7166.021} C_VEL
LIN {X 0,Y 626.651,Z 278.979,A -85,B 0,C 180,E1 -7168.308,E2 -7168.308} C_VEL
LIN {X 0,Y 626.662,Z 278.982,A -85,B 0,C 180,E1 -7171.274,E2 -7171.274} C_VEL
LIN {X 0,Y 626.613,Z 278.987,A -85,B 0,C 180,E1 -7173.44,E2 -7173.44} C_VEL
LIN {X 0,Y 626.661,Z 278.975,A -85,B 0,C 180,E1 -7176.273,E2 -7176.273} C_VEL
LIN {X 0,Y 626.643,Z 278.983,A -85,B 0,C 180,E1 -7179.042,E2 -7179.042} C_VEL
LIN {X 0,Y 626.674,Z 278.98,A -85,B 0,C 180,E1 -7181.808,E2 -7181.808} C_VEL
LIN {X 0,Y 626.684,Z 278.974,A -85,B 0,C 180,E1 -7184.44,E2 -7184.44} C_VEL
LIN {X 0,Y 626.699,Z 278.974,A -85,B 0,C 180,E1 -7187.083,E2 -7187.083} C_VEL
LIN {X 0,Y 626.667,Z 278.978,A -85,B 0,C 180,E1 -7189.698,E2 -7189.698} C_VEL
LIN {X 0,Y 626.726,Z 278.967,A -85,B 0,C 180,E1 -7192.293,E2 -7192.293} C_VEL
LIN {X 0,Y 626.767,Z 278.969,A -85,B 0,C 180,E1 -7194.871,E2 -7194.871} C_VEL
LIN {X 0,Y 626.756,Z 278.965,A -85,B 0,C 180,E1 -7198.079,E2 -7198.079} C_VEL
LIN {X 0,Y 626.82,Z 278.957,A -85,B 0,C 180,E1 -7200,E2 -7200} C_VEL
LIN {X 0,Y 626.784,Z 278.956,A -85,B 0,C 180,E1 -7201.921,E2 -7201.921} C_VEL
LIN {X 0,Y 626.784,Z 278.969,A -85,B 0,C 180,E1 -7205.129,E2 -7205.129} C_VEL
LIN {X 0,Y 626.728,Z 278.965,A -85,B 0,C 180,E1 -7207.707,E2 -7207.707} C_VEL
LIN {X 0,Y 626.753,Z 278.968,A -85,B 0,C 180,E1 -7210.447,E2 -7210.447} C_VEL
LIN {X 0,Y 626.698,Z 278.971,A -85,B 0,C 180,E1 -7213.575,E2 -7213.575} C_VEL
LIN {X 0,Y 626.676,Z 278.976,A -85,B 0,C 180,E1 -7216.226,E2 -7216.226} C_VEL
LIN {X 0,Y 626.652,Z 278.986,A -85,B 0,C 180,E1 -7218.914,E2 -7218.914} C_VEL
LIN {X 0,Y 626.66,Z 278.974,A -85,B 0,C 180,E1 -7221.645,E2 -7221.645} C_VEL
LIN {X 0,Y 626.669,Z 278.983,A -85,B 0,C 180,E1 -7224.429,E2 -7224.429} C_VEL
LIN {X 0,Y 626.634,Z 278.981,A -85,B 0,C 180,E1 -7227.277,E2 -7227.277} C_VEL
LIN {X 0,Y 626.657,Z 278.977,A -85,B 0,C 180,E1 -7229.46,E2 -7229.46} C_VEL
LIN {X 0,Y 626.642,Z 278.981,A -85,B 0,C 180,E1 -7231.846,E2 -7231.846} C_VEL
LIN {X 0,Y 626.662,Z 278.971,A -85,B 0,C 180,E1 -7234.754,E2 -7234.754} C_VEL
LIN {X 0,Y 626.68,Z 278.972,A -85,B 0,C 180,E1 -7237.483,E2 -7237.483} C_VEL
LIN {X 0,Y 626.648,Z 278.986,A -85,B 0,C 180,E1 -7240.532,E2 -7240.532} C_VEL
LIN {X 0,Y 626.66,Z 278.978,A -85,B 0,C 180,E1 -7242.986,E2 -7242.986} C_VEL
LIN {X 0,Y 626.631,Z 278.982,A -85,B 0,C 180,E1 -7245.675,E2 -7245.675} C_VEL
LIN {X 0,Y 626.682,Z 278.98,A -85,B 0,C 180,E1 -7247.888,E2 -7247.888} C_VEL
LIN {X 0,Y 626.645,Z 278.985,A -85,B 0,C 180,E1 -7250.467,E2 -7250.467} C_VEL
LIN {X 0,Y 626.671,Z 278.977,A -85,B 0,C 180,E1 -7252.877,E2 -7252.877} C_VEL
LIN {X 0,Y 626.654,Z 278.983,A -85,B 0,C 180,E1 -7255.249,E2 -7255.249} C_VEL
LIN {X 0,Y 626.644,Z 278.992,A -85,B 0,C 180,E1 -7258.158,E2 -7258.158} C_VEL
LIN {X 0,Y 626.671,Z 278.98,A -85,B 0,C 180,E1 -7260.671,E2 -7260.671} C_VEL
LIN {X 0,Y 626.648,Z 278.984,A -85,B 0,C 180,E1 -7262.726,E2 -7262.726} C_VEL
LIN {X 0,Y 626.666,Z 279.082,A -85,B 0,C 180,E1 -7264.419,E2 -7264.419} C_VEL
LIN {X 0,Y 629.176,Z 291.504,A -85,B 0,C 180,E1 -7266.049,E2 -7266.049} C_VEL
LIN {X 0,Y 628.912,Z 302.804,A -85,B 0,C 180,E1 -7267.411,E2 -7267.411} C_VEL
LIN {X 0,Y 628.282,Z 320.939,A -85,B 0,C 180,E1 -7269.563,E2 -7269.563} C_VEL
LIN {X 0,Y 627.664,Z 342.875,A -85,B 0,C 180,E1 -7272.13,E2 -7272.13} C_VEL
LIN {X 0,Y 627.132,Z 365.175,A -85,B 0,C 180,E1 -7274.681,E2 -7274.681} C_VEL
LIN {X 0,Y 629.591,Z 384.411,A -85,B 0,C 180,E1 -7274.97,E2 -7274.97} C_VEL
LIN {X 0,Y 628.923,Z 503.461,A -85,B 0,C 180,E1 -7276.353,E2 -7276.353} C_VEL
LIN {X 0,Y 628.589,Z 517.951,A -85,B 0,C 180,E1 -7276.653,E2 -7276.653} C_VEL
LIN {X 0,Y 628.24,Z 531.859,A -85,B 0,C 180,E1 -7277.076,E2 -7277.076} C_VEL
LIN {X 0,Y 627.832,Z 544.831,A -85,B 0,C 180,E1 -7277.6,E2 -7277.6} C_VEL
LIN {X 0,Y 627.425,Z 557.43,A -85,B 0,C 180,E1 -7278.246,E2 -7278.246} C_VEL
LIN {X 0,Y 627.105,Z 568.938,A -85,B 0,C 180,E1 -7278.974,E2 -7278.974} C_VEL
LIN {X 0,Y 626.765,Z 580.506,A -85,B 0,C 180,E1 -7279.864,E2 -7279.864} C_VEL
LIN {X 0,Y 626.41,Z 590.871,A -85,B 0,C 180,E1 -7280.833,E2 -7280.833} C_VEL
LIN {X 0,Y 626.134,Z 599.445,A -85,B 0,C 180,E1 -7281.802,E2 -7281.802} C_VEL
LIN {X 0,Y 625.971,Z 607.661,A -85,B 0,C 180,E1 -7282.931,E2 -7282.931} C_VEL
LIN {X 0,Y 625.894,Z 613.439,A -85,B 0,C 180,E1 -7283.899,E2 -7283.899} C_VEL
LIN {X 0,Y 625.828,Z 618.538,A -85,B 0,C 180,E1 -7284.947,E2 -7284.947} C_VEL
LIN {X 0,Y 625.819,Z 623.094,A -85,B 0,C 180,E1 -7286.151,E2 -7286.151} C_VEL
LIN {X 0,Y 625.802,Z 626.59,A -85,B 0,C 180,E1 -7287.436,E2 -7287.436} C_VEL
LIN {X 0,Y 625.805,Z 628.605,A -85,B 0,C 180,E1 -7288.719,E2 -7288.719} C_VEL
LIN {X 0,Y 625.788,Z 629.33,A -85,B 0,C 180,E1 -7290.002,E2 -7290.002} C_VEL
LIN {X 0,Y 625.805,Z 628.625,A -85,B 0,C 180,E1 -7291.284,E2 -7291.284} C_VEL
LIN {X 0,Y 625.805,Z 626.531,A -85,B 0,C 180,E1 -7292.568,E2 -7292.568} C_VEL
LIN {X 0,Y 625.82,Z 623.099,A -85,B 0,C 180,E1 -7293.852,E2 -7293.852} C_VEL
LIN {X 0,Y 625.832,Z 618.19,A -85,B 0,C 180,E1 -7295.138,E2 -7295.138} C_VEL
LIN {X 0,Y 625.936,Z 611.633,A -85,B 0,C 180,E1 -7296.427,E2 -7296.427} C_VEL
LIN {X 0,Y 626.035,Z 604.337,A -85,B 0,C 180,E1 -7297.556,E2 -7297.556} C_VEL
LIN {X 0,Y 626.268,Z 595.325,A -85,B 0,C 180,E1 -7298.686,E2 -7298.686} C_VEL
LIN {X 0,Y 626.52,Z 585.868,A -85,B 0,C 180,E1 -7299.655,E2 -7299.655} C_VEL
LIN {X 0,Y 626.854,Z 576.231,A -85,B 0,C 180,E1 -7300.482,E2 -7300.482} C_VEL
LIN {X 0,Y 627.157,Z 565.189,A -85,B 0,C 180,E1 -7301.272,E2 -7301.272} C_VEL
LIN {X 0,Y 627.529,Z 552.724,A -85,B 0,C 180,E1 -7302,E2 -7302} C_VEL
LIN {X 0,Y 627.95,Z 540.73,A -85,B 0,C 180,E1 -7302.564,E2 -7302.564} C_VEL
LIN {X 0,Y 628.258,Z 527.597,A -85,B 0,C 180,E1 -7303.049,E2 -7303.049} C_VEL
LIN {X 0,Y 628.628,Z 513.435,A -85,B 0,C 180,E1 -7303.431,E2 -7303.431} C_VEL
LIN {X 0,Y 628.869,Z 498.437,A -85,B 0,C 180,E1 -7303.692,E2 -7303.692} C_VEL
LIN {X 0,Y 629.463,Z 383.548,A -85,B 0,C 180,E1 -7305.008,E2 -7305.008} C_VEL
LIN {X 0,Y 627.091,Z 365.102,A -85,B 0,C 180,E1 -7305.281,E2 -7305.281} C_VEL
LIN {X 0,Y 627.68,Z 341.029,A -85,B 0,C 180,E1 -7308.041,E2 -7308.041} C_VEL
LIN {X 0,Y 628.353,Z 316.318,A -85,B 0,C 180,E1 -7310.9,E2 -7310.9} C_VEL
LIN {X 0,Y 629.095,Z 293.014,A -85,B 0,C 180,E1 -7313.631,E2 -7313.631} C_VEL
LIN {X 0,Y 628.318,Z 287.104,A -85,B 0,C 180,E1 -7314.362,E2 -7314.362} C_VEL
LIN {X 0,Y 626.654,Z 278.987,A -85,B 0,C 180,E1 -7315.417,E2 -7315.417} C_VEL
LIN {X 0,Y 626.653,Z 278.986,A -85,B 0,C 180,E1 -7318,E2 -7318} C_VEL
LIN {X 0,Y 626.611,Z 278.986,A -85,B 0,C 180,E1 -7320.601,E2 -7320.601} C_VEL
LIN {X 0,Y 626.633,Z 278.984,A -85,B 0,C 180,E1 -7323.212,E2 -7323.212} C_VEL
LIN {X 0,Y 626.623,Z 278.992,A -85,B 0,C 180,E1 -7325.54,E2 -7325.54} C_VEL
LIN {X 0,Y 626.627,Z 278.987,A -85,B 0,C 180,E1 -7327.938,E2 -7327.938} C_VEL
LIN {X 0,Y 626.614,Z 278.985,A -85,B 0,C 180,E1 -7330.525,E2 -7330.525} C_VEL
LIN {X 0,Y 626.639,Z 278.988,A -85,B 0,C 180,E1 -7333.401,E2 -7333.401} C_VEL
LIN {X 0,Y 626.636,Z 278.982,A -85,B 0,C 180,E1 -7336.13,E2 -7336.13} C_VEL
LIN {X 0,Y 626.621,Z 278.989,A -85,B 0,C 180,E1 -7338.738,E2 -7338.738} C_VEL
LIN {X 0,Y 626.631,Z 278.985,A -85,B 0,C 180,E1 -7341.487,E2 -7341.487} C_VEL
LIN {X 0,Y 626.678,Z 278.977,A -85,B 0,C 180,E1 -7343.673,E2 -7343.673} C_VEL
LIN {X 0,Y 626.634,Z 278.983,A -85,B 0,C 180,E1 -7346.021,E2 -7346.021} C_VEL
LIN {X 0,Y 626.676,Z 278.982,A -85,B 0,C 180,E1 -7348.31,E2 -7348.31} C_VEL
LIN {X 0,Y 626.66,Z 278.979,A -85,B 0,C 180,E1 -7351.273,E2 -7351.273} C_VEL
LIN {X 0,Y 626.625,Z 278.984,A -85,B 0,C 180,E1 -7353.441,E2 -7353.441} C_VEL
LIN {X 0,Y 626.683,Z 278.979,A -85,B 0,C 180,E1 -7355.572,E2 -7355.572} C_VEL
LIN {X 0,Y 626.69,Z 278.987,A -85,B 0,C 180,E1 -7358.356,E2 -7358.356} C_VEL
LIN {X 0,Y 626.663,Z 278.983,A -85,B 0,C 180,E1 -7361.086,E2 -7361.086} C_VEL
LIN {X 0,Y 626.707,Z 278.981,A -85,B 0,C 180,E1 -7363.987,E2 -7363.987} C_VEL
LIN {X 0,Y 626.703,Z 278.979,A -85,B 0,C 180,E1 -7366.502,E2 -7366.502} C_VEL
LIN {X 0,Y 626.748,Z 279.156,A -85,B 0,C 180,E1 -7369.077,E2 -7369.077} C_VEL
LIN {X 0,Y 628.293,Z 288.121,A -85,B 0,C 180,E1 -7370.211,E2 -7370.211} C_VEL
LIN {X 0,Y 628.106,Z 309.404,A -85,B 0,C 180,E1 -7372.793,E2 -7372.793} C_VEL
LIN {X 0,Y 627.612,Z 330.58,A -85,B 0,C 180,E1 -7375.359,E2 -7375.359} C_VEL
LIN {X 0,Y 627.528,Z 341.876,A -85,B 0,C 180,E1 -7376.741,E2 -7376.741} C_VEL
LIN {X 0,Y 629.71,Z 355.606,A -85,B 0,C 180,E1 -7376.991,E2 -7376.991} C_VEL
LIN {X 0,Y 628.65,Z 479.798,A -85,B 0,C 180,E1 -7378.543,E2 -7378.543} C_VEL
LIN {X 0,Y 628.404,Z 494.755,A -85,B 0,C 180,E1 -7378.862,E2 -7378.862} C_VEL
LIN {X 0,Y 628.094,Z 509.253,A -85,B 0,C 180,E1 -7379.321,E2 -7379.321} C_VEL
LIN {X 0,Y 627.813,Z 520.023,A -85,B 0,C 180,E1 -7379.76,E2 -7379.76} C_VEL
LIN {X 0,Y 627.447,Z 532.568,A -85,B 0,C 180,E1 -7380.4,E2 -7380.4} C_VEL
LIN {X 0,Y 627.196,Z 545.126,A -85,B 0,C 180,E1 -7381.2,E2 -7381.2} C_VEL
LIN {X 0,Y 626.784,Z 556.456,A -85,B 0,C 180,E1 -7382.081,E2 -7382.081} C_VEL
LIN {X 0,Y 626.49,Z 566.623,A -85,B 0,C 180,E1 -7383.044,E2 -7383.044} C_VEL
LIN {X 0,Y 626.174,Z 575.057,A -85,B 0,C 180,E1 -7384.009,E2 -7384.009} C_VEL
LIN {X 0,Y 626.072,Z 583.116,A -85,B 0,C 180,E1 -7385.135,E2 -7385.135} C_VEL
LIN {X 0,Y 625.972,Z 588.768,A -85,B 0,C 180,E1 -7386.102,E2 -7386.102} C_VEL
LIN {X 0,Y 625.858,Z 593.392,A -85,B 0,C 180,E1 -7387.072,E2 -7387.072} C_VEL
LIN {X 0,Y 625.759,Z 598.179,A -85,B 0,C 180,E1 -7388.367,E2 -7388.367} C_VEL
LIN {X 0,Y 625.763,Z 601.437,A -85,B 0,C 180,E1 -7389.666,E2 -7389.666} C_VEL
LIN {X 0,Y 625.655,Z 603.252,A -85,B 0,C 180,E1 -7390.972,E2 -7390.972} C_VEL
LIN {X 0,Y 625.685,Z 603.674,A -85,B 0,C 180,E1 -7392.281,E2 -7392.281} C_VEL
LIN {X 0,Y 625.705,Z 602.695,A -85,B 0,C 180,E1 -7393.597,E2 -7393.597} C_VEL
LIN {X 0,Y 625.73,Z 600.282,A -85,B 0,C 180,E1 -7394.92,E2 -7394.92} C_VEL
LIN {X 0,Y 625.818,Z 596.348,A -85,B 0,C 180,E1 -7396.249,E2 -7396.249} C_VEL
LIN {X 0,Y 625.885,Z 592.265,A -85,B 0,C 180,E1 -7397.252,E2 -7397.252} C_VEL
LIN {X 0,Y 625.977,Z 587.141,A -85,B 0,C 180,E1 -7398.259,E2 -7398.259} C_VEL
LIN {X 0,Y 626.138,Z 579.698,A -85,B 0,C 180,E1 -7399.439,E2 -7399.439} C_VEL
LIN {X 0,Y 626.363,Z 571.802,A -85,B 0,C 180,E1 -7400.454,E2 -7400.454} C_VEL
LIN {X 0,Y 626.636,Z 562.184,A -85,B 0,C 180,E1 -7401.474,E2 -7401.474} C_VEL
LIN {X 0,Y 626.961,Z 551.392,A -85,B 0,C 180,E1 -7402.411,E2 -7402.411} C_VEL
LIN {X 0,Y 627.352,Z 539.394,A -85,B 0,C 180,E1 -7403.264,E2 -7403.264} C_VEL
LIN {X 0,Y 627.644,Z 527.583,A -85,B 0,C 180,E1 -7403.95,E2 -7403.95} C_VEL
LIN {X 0,Y 627.984,Z 514.727,A -85,B 0,C 180,E1 -7404.55,E2 -7404.55} C_VEL
LIN {X 0,Y 628.312,Z 501.756,A -85,B 0,C 180,E1 -7405.02,E2 -7405.02} C_VEL
LIN {X 0,Y 628.563,Z 487.603,A -85,B 0,C 180,E1 -7405.395,E2 -7405.395} C_VEL
LIN {X 0,Y 628.751,Z 472.946,A -85,B 0,C 180,E1 -7405.646,E2 -7405.646} C_VEL
LIN {X 0,Y 629.505,Z 354.638,A -85,B 0,C 180,E1 -7407.082,E2 -7407.082} C_VEL
LIN {X 0,Y 627.367,Z 341.398,A -85,B 0,C 180,E1 -7407.31,E2 -7407.31} C_VEL
LIN {X 0,Y 627.785,Z 320.108,A -85,B 0,C 180,E1 -7409.958,E2 -7409.958} C_VEL
LIN {X 0,Y 628.149,Z 300.775,A -85,B 0,C 180,E1 -7412.36,E2 -7412.36} C_VEL
LIN {X 0,Y 628.356,Z 288.657,A -85,B 0,C 180,E1 -7413.874,E2 -7413.874} C_VEL
LIN {X 0,Y 626.665,Z 278.984,A -85,B 0,C 180,E1 -7415.136,E2 -7415.136} C_VEL
LIN {X 0,Y 626.668,Z 278.98,A -85,B 0,C 180,E1 -7417.477,E2 -7417.477} C_VEL
LIN {X 0,Y 626.651,Z 278.985,A -85,B 0,C 180,E1 -7418.491,E2 -7418.491} C_VEL
LIN {X 0,Y 626.014,Z 279.067,A -85,B 0,C 180,E1 -7419.028,E2 -7419.028} C_VEL
LIN {X 0,Y 623.144,Z 279.423,A -85,B 0,C 180,E1 -7419.897,E2 -7419.897} C_VEL
LIN {X 0,Y 620.699,Z 279.725,A -85,B 0,C 180,E1 -7420.597,E2 -7420.597} C_VEL
LIN {X 0,Y 619.649,Z 279.853,A -85,B 0,C 180,E1 -7421.137,E2 -7421.137} C_VEL
LIN {X 0,Y 619.565,Z 279.863,A -85,B 0,C 180,E1 -7421.319,E2 -7421.319} C_VEL
LIN {X 0,Y 619.595,Z 279.863,A -85,B 0,C 180,E1 -7423.654,E2 -7423.654} C_VEL
LIN {X 0,Y 619.594,Z 279.862,A -85,B 0,C 180,E1 -7426.4,E2 -7426.4} C_VEL
LIN {X 0,Y 619.576,Z 279.866,A -85,B 0,C 180,E1 -7429.24,E2 -7429.24} C_VEL
LIN {X 0,Y 619.582,Z 279.866,A -85,B 0,C 180,E1 -7431.552,E2 -7431.552} C_VEL
LIN {X 0,Y 619.61,Z 279.861,A -85,B 0,C 180,E1 -7433.995,E2 -7433.995} C_VEL
LIN {X 0,Y 619.59,Z 279.864,A -85,B 0,C 180,E1 -7436.779,E2 -7436.779} C_VEL
LIN {X 0,Y 619.615,Z 279.863,A -85,B 0,C 180,E1 -7439.421,E2 -7439.421} C_VEL
LIN {X 0,Y 619.598,Z 279.862,A -85,B 0,C 180,E1 -7442.386,E2 -7442.386} C_VEL
LIN {X 0,Y 619.618,Z 279.861,A -85,B 0,C 180,E1 -7445.274,E2 -7445.274} C_VEL
LIN {X 0,Y 619.668,Z 279.853,A -85,B 0,C 180,E1 -7448.097,E2 -7448.097} C_VEL
LIN {X 0,Y 619.634,Z 279.858,A -85,B 0,C 180,E1 -7450.862,E2 -7450.862} C_VEL
LIN {X 0,Y 619.643,Z 279.854,A -85,B 0,C 180,E1 -7453.583,E2 -7453.583} C_VEL
LIN {X 0,Y 619.672,Z 279.854,A -85,B 0,C 180,E1 -7456.433,E2 -7456.433} C_VEL
LIN {X 0,Y 619.696,Z 279.849,A -85,B 0,C 180,E1 -7459.579,E2 -7459.579} C_VEL
LIN {X 0,Y 619.694,Z 279.854,A -85,B 0,C 180,E1 -7462.203,E2 -7462.203} C_VEL
LIN {X 0,Y 619.741,Z 279.857,A -85,B 0,C 180,E1 -7463.731,E2 -7463.731} C_VEL
LIN {X 0,Y 620.516,Z 286.11,A -85,B 0,C 180,E1 -7464.817,E2 -7464.817} C_VEL
LIN {X 0,Y 620.34,Z 296.998,A -85,B 0,C 180,E1 -7466.641,E2 -7466.641} C_VEL
LIN {X 0,Y 622.881,Z 309.45,A -85,B 0,C 180,E1 -7466.856,E2 -7466.856} C_VEL
LIN {X 0,Y 622.052,Z 432.043,A -85,B 0,C 180,E1 -7468.284,E2 -7468.284} C_VEL
LIN {X 0,Y 621.915,Z 446.516,A -85,B 0,C 180,E1 -7468.587,E2 -7468.587} C_VEL
LIN {X 0,Y 621.67,Z 459.8,A -85,B 0,C 180,E1 -7468.99,E2 -7468.99} C_VEL
LIN {X 0,Y 621.368,Z 471.07,A -85,B 0,C 180,E1 -7469.433,E2 -7469.433} C_VEL
LIN {X 0,Y 621.054,Z 483.945,A -85,B 0,C 180,E1 -7470.079,E2 -7470.079} C_VEL
LIN {X 0,Y 620.595,Z 495.674,A -85,B 0,C 180,E1 -7470.807,E2 -7470.807} C_VEL
LIN {X 0,Y 620.287,Z 506.366,A -85,B 0,C 180,E1 -7471.616,E2 -7471.616} C_VEL
LIN {X 0,Y 619.843,Z 516.982,A -85,B 0,C 180,E1 -7472.589,E2 -7472.589} C_VEL
LIN {X 0,Y 619.591,Z 525.74,A -85,B 0,C 180,E1 -7473.563,E2 -7473.563} C_VEL
LIN {X 0,Y 619.249,Z 534.168,A -85,B 0,C 180,E1 -7474.702,E2 -7474.702} C_VEL
LIN {X 0,Y 619.142,Z 540.953,A -85,B 0,C 180,E1 -7475.842,E2 -7475.842} C_VEL
LIN {X 0,Y 618.987,Z 545.665,A -85,B 0,C 180,E1 -7476.822,E2 -7476.822} C_VEL
LIN {X 0,Y 618.822,Z 550.552,A -85,B 0,C 180,E1 -7478.132,E2 -7478.132} C_VEL
LIN {X 0,Y 618.801,Z 553.228,A -85,B 0,C 180,E1 -7479.116,E2 -7479.116} C_VEL
LIN {X 0,Y 618.734,Z 555.575,A -85,B 0,C 180,E1 -7480.434,E2 -7480.434} C_VEL
LIN {X 0,Y 618.688,Z 556.57,A -85,B 0,C 180,E1 -7481.757,E2 -7481.757} C_VEL
LIN {X 0,Y 618.769,Z 556.21,A -85,B 0,C 180,E1 -7483.083,E2 -7483.083} C_VEL
LIN {X 0,Y 618.755,Z 554.486,A -85,B 0,C 180,E1 -7484.419,E2 -7484.419} C_VEL
LIN {X 0,Y 618.877,Z 551.327,A -85,B 0,C 180,E1 -7485.759,E2 -7485.759} C_VEL
LIN {X 0,Y 618.959,Z 547.896,A -85,B 0,C 180,E1 -7486.77,E2 -7486.77} C_VEL
LIN {X 0,Y 619.06,Z 543.54,A -85,B 0,C 180,E1 -7487.786,E2 -7487.786} C_VEL
LIN {X 0,Y 619.315,Z 537.112,A -85,B 0,C 180,E1 -7488.973,E2 -7488.973} C_VEL
LIN {X 0,Y 619.506,Z 530.082,A -85,B 0,C 180,E1 -7490.025,E2 -7490.025} C_VEL
LIN {X 0,Y 619.838,Z 521.984,A -85,B 0,C 180,E1 -7491.024,E2 -7491.024} C_VEL
LIN {X 0,Y 620.211,Z 512.615,A -85,B 0,C 180,E1 -7491.984,E2 -7491.984} C_VEL
LIN {X 0,Y 620.569,Z 501.608,A -85,B 0,C 180,E1 -7492.915,E2 -7492.915} C_VEL
LIN {X 0,Y 620.978,Z 490.434,A -85,B 0,C 180,E1 -7493.691,E2 -7493.691} C_VEL
LIN {X 0,Y 621.327,Z 478.719,A -85,B 0,C 180,E1 -7494.358,E2 -7494.358} C_VEL
LIN {X 0,Y 621.691,Z 465.758,A -85,B 0,C 180,E1 -7494.946,E2 -7494.946} C_VEL
LIN {X 0,Y 622.013,Z 453.02,A -85,B 0,C 180,E1 -7495.39,E2 -7495.39} C_VEL
LIN {X 0,Y 622.174,Z 439.499,A -85,B 0,C 180,E1 -7495.737,E2 -7495.737} C_VEL
LIN {X 0,Y 622.267,Z 425.513,A -85,B 0,C 180,E1 -7495.965,E2 -7495.965} C_VEL
LIN {X 0,Y 623.026,Z 309.363,A -85,B 0,C 180,E1 -7497.317,E2 -7497.317} C_VEL
LIN {X 0,Y 620.521,Z 297.247,A -85,B 0,C 180,E1 -7497.549,E2 -7497.549} C_VEL
LIN {X 0,Y 620.713,Z 286.827,A -85,B 0,C 180,E1 -7499.328,E2 -7499.328} C_VEL
LIN {X 0,Y 619.606,Z 279.866,A -85,B 0,C 180,E1 -7500.576,E2 -7500.576} C_VEL
LIN {X 0,Y 619.572,Z 279.863,A -85,B 0,C 180,E1 -7503.218,E2 -7503.218} C_VEL
LIN {X 0,Y 619.609,Z 279.866,A -85,B 0,C 180,E1 -7506.001,E2 -7506.001} C_VEL
LIN {X 0,Y 619.599,Z 279.859,A -85,B 0,C 180,E1 -7508.737,E2 -7508.737} C_VEL
LIN {X 0,Y 619.561,Z 279.865,A -85,B 0,C 180,E1 -7511.741,E2 -7511.741} C_VEL
LIN {X 0,Y 619.568,Z 279.858,A -85,B 0,C 180,E1 -7514.583,E2 -7514.583} C_VEL
LIN {X 0,Y 619.588,Z 279.861,A -85,B 0,C 180,E1 -7517.289,E2 -7517.289} C_VEL
LIN {X 0,Y 619.579,Z 279.868,A -85,B 0,C 180,E1 -7519.88,E2 -7519.88} C_VEL
LIN {X 0,Y 619.609,Z 279.857,A -85,B 0,C 180,E1 -7522.378,E2 -7522.378} C_VEL
LIN {X 0,Y 619.589,Z 279.85,A -85,B 0,C 180,E1 -7524.791,E2 -7524.791} C_VEL
LIN {X 0,Y 619.567,Z 279.863,A -85,B 0,C 180,E1 -7527.135,E2 -7527.135} C_VEL
LIN {X 0,Y 619.628,Z 279.857,A -85,B 0,C 180,E1 -7529.423,E2 -7529.423} C_VEL
LIN {X 0,Y 619.624,Z 279.858,A -85,B 0,C 180,E1 -7531.848,E2 -7531.848} C_VEL
LIN {X 0,Y 619.567,Z 279.862,A -85,B 0,C 180,E1 -7534.741,E2 -7534.741} C_VEL
LIN {X 0,Y 619.613,Z 279.859,A -85,B 0,C 180,E1 -7537.396,E2 -7537.396} C_VEL
LIN {X 0,Y 619.618,Z 279.853,A -85,B 0,C 180,E1 -7540.176,E2 -7540.176} C_VEL
LIN {X 0,Y 619.594,Z 279.859,A -85,B 0,C 180,E1 -7542.907,E2 -7542.907} C_VEL
LIN {X 0,Y 619.624,Z 279.856,A -85,B 0,C 180,E1 -7544.93,E2 -7544.93} C_VEL
LIN {X 0,Y 619.663,Z 279.848,A -85,B 0,C 180,E1 -7546.934,E2 -7546.934} C_VEL
LIN {X 0,Y 619.666,Z 279.852,A -85,B 0,C 180,E1 -7549.58,E2 -7549.58} C_VEL
LIN {X 0,Y 619.682,Z 279.845,A -85,B 0,C 180,E1 -7552.204,E2 -7552.204} C_VEL
LIN {X 0,Y 619.712,Z 279.847,A -85,B 0,C 180,E1 -7554.812,E2 -7554.812} C_VEL
LIN {X 0,Y 619.553,Z 279.861,A -85,B 0,C 180,E1 -7556.759,E2 -7556.759} C_VEL
LIN {X 0,Y 619.844,Z 279.833,A -85,B 0,C 180,E1 -7559.353,E2 -7559.353} C_VEL
LIN {X 0,Y 619.841,Z 279.827,A -85,B 0,C 180,E1 -7561.295,E2 -7561.295} C_VEL
LIN {X 0,Y 619.731,Z 279.843,A -85,B 0,C 180,E1 -7564.538,E2 -7564.538} C_VEL
LIN {X 0,Y 619.699,Z 279.846,A -85,B 0,C 180,E1 -7567.142,E2 -7567.142} C_VEL
LIN {X 0,Y 619.722,Z 279.845,A -85,B 0,C 180,E1 -7570.493,E2 -7570.493} C_VEL
LIN {X 0,Y 619.66,Z 279.847,A -85,B 0,C 180,E1 -7573.732,E2 -7573.732} C_VEL
LIN {X 0,Y 619.646,Z 279.854,A -85,B 0,C 180,E1 -7576.415,E2 -7576.415} C_VEL
LIN {X 0,Y 619.617,Z 279.858,A -85,B 0,C 180,E1 -7579.137,E2 -7579.137} C_VEL
LIN {X 0,Y 619.62,Z 279.852,A -85,B 0,C 180,E1 -7582.04,E2 -7582.04} C_VEL
LIN {X 0,Y 619.598,Z 279.865,A -85,B 0,C 180,E1 -7584.726,E2 -7584.726} C_VEL
LIN {X 0,Y 619.593,Z 279.857,A -85,B 0,C 180,E1 -7587.613,E2 -7587.613} C_VEL
LIN {X 0,Y 619.591,Z 279.858,A -85,B 0,C 180,E1 -7589.829,E2 -7589.829} C_VEL
LIN {X 0,Y 619.606,Z 279.86,A -85,B 0,C 180,E1 -7592.095,E2 -7592.095} C_VEL
LIN {X 0,Y 619.614,Z 279.855,A -85,B 0,C 180,E1 -7594.418,E2 -7594.418} C_VEL
LIN {X 0,Y 619.628,Z 279.854,A -85,B 0,C 180,E1 -7596.807,E2 -7596.807} C_VEL
LIN {X 0,Y 619.605,Z 279.857,A -85,B 0,C 180,E1 -7599.277,E2 -7599.277} C_VEL
LIN {X 0,Y 619.599,Z 279.861,A -85,B 0,C 180,E1 -7601.835,E2 -7601.835} C_VEL
LIN {X 0,Y 619.58,Z 279.863,A -85,B 0,C 180,E1 -7604.587,E2 -7604.587} C_VEL
LIN {X 0,Y 619.655,Z 279.85,A -85,B 0,C 180,E1 -7607.298,E2 -7607.298} C_VEL
LIN {X 0,Y 619.588,Z 279.868,A -85,B 0,C 180,E1 -7610.241,E2 -7610.241} C_VEL
LIN {X 0,Y 619.65,Z 279.857,A -85,B 0,C 180,E1 -7612.384,E2 -7612.384} C_VEL
LIN {X 0,Y 619.63,Z 279.859,A -85,B 0,C 180,E1 -7614.797,E2 -7614.797} C_VEL
LIN {X 0,Y 619.597,Z 279.862,A -85,B 0,C 180,E1 -7617.14,E2 -7617.14} C_VEL
LIN {X 0,Y 619.641,Z 279.86,A -85,B 0,C 180,E1 -7619.426,E2 -7619.426} C_VEL
LIN {X 0,Y 619.638,Z 279.862,A -85,B 0,C 180,E1 -7621.851,E2 -7621.851} C_VEL
LIN {X 0,Y 619.632,Z 280.045,A -85,B 0,C 180,E1 -7624.248,E2 -7624.248} C_VEL
LIN {X 0,Y 622.21,Z 292.504,A -85,B 0,C 180,E1 -7625.91,E2 -7625.91} C_VEL
LIN {X 0,Y 622.193,Z 299.709,A -85,B 0,C 180,E1 -7626.797,E2 -7626.797} C_VEL
LIN {X 0,Y 621.31,Z 322.563,A -85,B 0,C 180,E1 -7629.546,E2 -7629.546} C_VEL
LIN {X 0,Y 620.666,Z 344.041,A -85,B 0,C 180,E1 -7632.092,E2 -7632.092} C_VEL
LIN {X 0,Y 620.15,Z 364.463,A -85,B 0,C 180,E1 -7634.484,E2 -7634.484} C_VEL
LIN {X 0,Y 622.756,Z 385.033,A -85,B 0,C 180,E1 -7634.801,E2 -7634.801} C_VEL
LIN {X 0,Y 622.059,Z 502.448,A -85,B 0,C 180,E1 -7636.179,E2 -7636.179} C_VEL
LIN {X 0,Y 621.713,Z 517.138,A -85,B 0,C 180,E1 -7636.482,E2 -7636.482} C_VEL
LIN {X 0,Y 621.322,Z 530.572,A -85,B 0,C 180,E1 -7636.888,E2 -7636.888} C_VEL
LIN {X 0,Y 620.89,Z 544.604,A -85,B 0,C 180,E1 -7637.459,E2 -7637.459} C_VEL
LIN {X 0,Y 620.437,Z 557.154,A -85,B 0,C 180,E1 -7638.112,E2 -7638.112} C_VEL
LIN {X 0,Y 620.069,Z 568.632,A -85,B 0,C 180,E1 -7638.848,E2 -7638.848} C_VEL
LIN {X 0,Y 619.796,Z 578.22,A -85,B 0,C 180,E1 -7639.584,E2 -7639.584} C_VEL
LIN {X 0,Y 619.446,Z 587.257,A -85,B 0,C 180,E1 -7640.401,E2 -7640.401} C_VEL
LIN {X 0,Y 619.157,Z 596.357,A -85,B 0,C 180,E1 -7641.381,E2 -7641.381} C_VEL
LIN {X 0,Y 618.953,Z 605.08,A -85,B 0,C 180,E1 -7642.524,E2 -7642.524} C_VEL
LIN {X 0,Y 618.852,Z 611.226,A -85,B 0,C 180,E1 -7643.503,E2 -7643.503} C_VEL
LIN {X 0,Y 618.741,Z 617.84,A -85,B 0,C 180,E1 -7644.806,E2 -7644.806} C_VEL
LIN {X 0,Y 618.731,Z 622.897,A -85,B 0,C 180,E1 -7646.107,E2 -7646.107} C_VEL
LIN {X 0,Y 618.699,Z 626.415,A -85,B 0,C 180,E1 -7647.406,E2 -7647.406} C_VEL
LIN {X 0,Y 618.731,Z 628.486,A -85,B 0,C 180,E1 -7648.704,E2 -7648.704} C_VEL
LIN {X 0,Y 618.708,Z 629.185,A -85,B 0,C 180,E1 -7650.002,E2 -7650.002} C_VEL
LIN {X 0,Y 618.732,Z 628.482,A -85,B 0,C 180,E1 -7651.299,E2 -7651.299} C_VEL
LIN {X 0,Y 618.703,Z 626.371,A -85,B 0,C 180,E1 -7652.597,E2 -7652.597} C_VEL
LIN {X 0,Y 618.732,Z 622.825,A -85,B 0,C 180,E1 -7653.896,E2 -7653.896} C_VEL
LIN {X 0,Y 618.747,Z 617.784,A -85,B 0,C 180,E1 -7655.197,E2 -7655.197} C_VEL
LIN {X 0,Y 618.813,Z 613.012,A -85,B 0,C 180,E1 -7656.175,E2 -7656.175} C_VEL
LIN {X 0,Y 618.927,Z 606.134,A -85,B 0,C 180,E1 -7657.316,E2 -7657.316} C_VEL
LIN {X 0,Y 619.108,Z 597.599,A -85,B 0,C 180,E1 -7658.459,E2 -7658.459} C_VEL
LIN {X 0,Y 619.414,Z 588.705,A -85,B 0,C 180,E1 -7659.439,E2 -7659.439} C_VEL
LIN {X 0,Y 619.784,Z 577.939,A -85,B 0,C 180,E1 -7660.419,E2 -7660.419} C_VEL
LIN {X 0,Y 620.084,Z 567.051,A -85,B 0,C 180,E1 -7661.238,E2 -7661.238} C_VEL
LIN {X 0,Y 620.491,Z 555.153,A -85,B 0,C 180,E1 -7661.973,E2 -7661.973} C_VEL
LIN {X 0,Y 620.909,Z 542.027,A -85,B 0,C 180,E1 -7662.626,E2 -7662.626} C_VEL
LIN {X 0,Y 621.29,Z 528.192,A -85,B 0,C 180,E1 -7663.157,E2 -7663.157} C_VEL
LIN {X 0,Y 621.683,Z 513.52,A -85,B 0,C 180,E1 -7663.563,E2 -7663.563} C_VEL
LIN {X 0,Y 621.928,Z 498.823,A -85,B 0,C 180,E1 -7663.827,E2 -7663.827} C_VEL
LIN {X 0,Y 622.529,Z 383.92,A -85,B 0,C 180,E1 -7665.159,E2 -7665.159} C_VEL
LIN {X 0,Y 620.081,Z 364.586,A -85,B 0,C 180,E1 -7665.458,E2 -7665.458} C_VEL
LIN {X 0,Y 620.719,Z 339.073,A -85,B 0,C 180,E1 -7668.42,E2 -7668.42} C_VEL
LIN {X 0,Y 621.477,Z 312.9,A -85,B 0,C 180,E1 -7671.489,E2 -7671.489} C_VEL
LIN {X 0,Y 622.144,Z 293.957,A -85,B 0,C 180,E1 -7673.735,E2 -7673.735} C_VEL
LIN {X 0,Y 621.213,Z 287.762,A -85,B 0,C 180,E1 -7674.513,E2 -7674.513} C_VEL
LIN {X 0,Y 619.621,Z 279.863,A -85,B 0,C 180,E1 -7675.531,E2 -7675.531} C_VEL
LIN {X 0,Y 619.618,Z 279.861,A -85,B 0,C 180,E1 -7678.347,E2 -7678.347} C_VEL
LIN {X 0,Y 619.579,Z 279.865,A -85,B 0,C 180,E1 -7681.336,E2 -7681.336} C_VEL
LIN {X 0,Y 619.588,Z 279.868,A -85,B 0,C 180,E1 -7683.639,E2 -7683.639} C_VEL
LIN {X 0,Y 619.596,Z 279.859,A -85,B 0,C 180,E1 -7686.617,E2 -7686.617} C_VEL
LIN {X 0,Y 619.581,Z 279.869,A -85,B 0,C 180,E1 -7689.279,E2 -7689.279} C_VEL
LIN {X 0,Y 619.574,Z 279.863,A -85,B 0,C 180,E1 -7691.838,E2 -7691.838} C_VEL
LIN {X 0,Y 619.58,Z 279.862,A -85,B 0,C 180,E1 -7694.584,E2 -7694.584} C_VEL
LIN {X 0,Y 619.596,Z 279.866,A -85,B 0,C 180,E1 -7697.293,E2 -7697.293} C_VEL
LIN {X 0,Y 619.555,Z 279.864,A -85,B 0,C 180,E1 -7699.878,E2 -7699.878} C_VEL
LIN {X 0,Y 619.587,Z 279.863,A -85,B 0,C 180,E1 -7702.376,E2 -7702.376} C_VEL
LIN {X 0,Y 619.616,Z 279.864,A -85,B 0,C 180,E1 -7704.793,E2 -7704.793} C_VEL
LIN {X 0,Y 619.593,Z 279.862,A -85,B 0,C 180,E1 -7707.137,E2 -7707.137} C_VEL
LIN {X 0,Y 619.623,Z 279.856,A -85,B 0,C 180,E1 -7709.423,E2 -7709.423} C_VEL
LIN {X 0,Y 619.597,Z 279.867,A -85,B 0,C 180,E1 -7712.387,E2 -7712.387} C_VEL
LIN {X 0,Y 619.619,Z 279.858,A -85,B 0,C 180,E1 -7715.275,E2 -7715.275} C_VEL
LIN {X 0,Y 619.67,Z 279.862,A -85,B 0,C 180,E1 -7718.098,E2 -7718.098} C_VEL
LIN {X 0,Y 619.629,Z 279.86,A -85,B 0,C 180,E1 -7720.863,E2 -7720.863} C_VEL
LIN {X 0,Y 619.636,Z 279.861,A -85,B 0,C 180,E1 -7723.584,E2 -7723.584} C_VEL
LIN {X 0,Y 619.675,Z 279.855,A -85,B 0,C 180,E1 -7726.435,E2 -7726.435} C_VEL
LIN {X 0,Y 619.7,Z 280.046,A -85,B 0,C 180,E1 -7728.922,E2 -7728.922} C_VEL
LIN {X 0,Y 621.378,Z 289.234,A -85,B 0,C 180,E1 -7730.101,E2 -7730.101} C_VEL
LIN {X 0,Y 621.184,Z 310.564,A -85,B 0,C 180,E1 -7732.712,E2 -7732.712} C_VEL
LIN {X 0,Y 620.698,Z 334.528,A -85,B 0,C 180,E1 -7735.631,E2 -7735.631} C_VEL
LIN {X 0,Y 620.574,Z 342.097,A -85,B 0,C 180,E1 -7736.562,E2 -7736.562} C_VEL
LIN {X 0,Y 622.899,Z 356.265,A -85,B 0,C 180,E1 -7736.817,E2 -7736.817} C_VEL
LIN {X 0,Y 621.742,Z 480.652,A -85,B 0,C 180,E1 -7738.406,E2 -7738.406} C_VEL
LIN {X 0,Y 621.502,Z 495.319,A -85,B 0,C 180,E1 -7738.729,E2 -7738.729} C_VEL
LIN {X 0,Y 621.141,Z 509.704,A -85,B 0,C 180,E1 -7739.192,E2 -7739.192} C_VEL
LIN {X 0,Y 620.834,Z 521.256,A -85,B 0,C 180,E1 -7739.677,E2 -7739.677} C_VEL
LIN {X 0,Y 620.452,Z 533.586,A -85,B 0,C 180,E1 -7740.323,E2 -7740.323} C_VEL
LIN {X 0,Y 620.182,Z 545.988,A -85,B 0,C 180,E1 -7741.132,E2 -7741.132} C_VEL
LIN {X 0,Y 619.783,Z 556.253,A -85,B 0,C 180,E1 -7741.943,E2 -7741.943} C_VEL
LIN {X 0,Y 619.436,Z 566.481,A -85,B 0,C 180,E1 -7742.917,E2 -7742.917} C_VEL
LIN {X 0,Y 619.14,Z 574.965,A -85,B 0,C 180,E1 -7743.892,E2 -7743.892} C_VEL
LIN {X 0,Y 618.988,Z 582.863,A -85,B 0,C 180,E1 -7744.995,E2 -7744.995} C_VEL
LIN {X 0,Y 618.887,Z 589.619,A -85,B 0,C 180,E1 -7746.172,E2 -7746.172} C_VEL
LIN {X 0,Y 618.744,Z 595.413,A -85,B 0,C 180,E1 -7747.48,E2 -7747.48} C_VEL
LIN {X 0,Y 618.657,Z 598.745,A -85,B 0,C 180,E1 -7748.464,E2 -7748.464} C_VEL
LIN {X 0,Y 618.675,Z 601.825,A -85,B 0,C 180,E1 -7749.778,E2 -7749.778} C_VEL
LIN {X 0,Y 618.573,Z 603.501,A -85,B 0,C 180,E1 -7751.099,E2 -7751.099} C_VEL
LIN {X 0,Y 618.591,Z 603.782,A -85,B 0,C 180,E1 -7752.424,E2 -7752.424} C_VEL
LIN {X 0,Y 618.661,Z 603.334,A -85,B 0,C 180,E1 -7753.17,E2 -7753.17} C_VEL
LIN {X 0,Y 618.602,Z 601.556,A -85,B 0,C 180,E1 -7754.425,E2 -7754.425} C_VEL
LIN {X 0,Y 618.668,Z 600.081,A -85,B 0,C 180,E1 -7755.094,E2 -7755.094} C_VEL
LIN {X 0,Y 618.732,Z 595.912,A -85,B 0,C 180,E1 -7756.44,E2 -7756.44} C_VEL
LIN {X 0,Y 618.806,Z 591.71,A -85,B 0,C 180,E1 -7757.455,E2 -7757.455} C_VEL
LIN {X 0,Y 618.95,Z 585.409,A -85,B 0,C 180,E1 -7758.645,E2 -7758.645} C_VEL
LIN {X 0,Y 619.139,Z 577.429,A -85,B 0,C 180,E1 -7759.84,E2 -7759.84} C_VEL
LIN {X 0,Y 619.407,Z 569.001,A -85,B 0,C 180,E1 -7760.868,E2 -7760.868} C_VEL
LIN {X 0,Y 619.736,Z 558.732,A -85,B 0,C 180,E1 -7761.899,E2 -7761.899} C_VEL
LIN {X 0,Y 620.068,Z 547.13,A -85,B 0,C 180,E1 -7762.849,E2 -7762.849} C_VEL
LIN {X 0,Y 620.459,Z 535.566,A -85,B 0,C 180,E1 -7763.621,E2 -7763.621} C_VEL
LIN {X 0,Y 620.808,Z 522.675,A -85,B 0,C 180,E1 -7764.319,E2 -7764.319} C_VEL
LIN {X 0,Y 621.128,Z 509.492,A -85,B 0,C 180,E1 -7764.883,E2 -7764.883} C_VEL
LIN {X 0,Y 621.454,Z 495.469,A -85,B 0,C 180,E1 -7765.337,E2 -7765.337} C_VEL
LIN {X 0,Y 621.744,Z 481.457,A -85,B 0,C 180,E1 -7765.653,E2 -7765.653} C_VEL
LIN {X 0,Y 621.871,Z 456.617,A -85,B 0,C 180,E1 -7765.982,E2 -7765.982} C_VEL
LIN {X 0,Y 622.6,Z 355.2,A -85,B 0,C 180,E1 -7767.235,E2 -7767.235} C_VEL
LIN {X 0,Y 620.382,Z 341.479,A -85,B 0,C 180,E1 -7767.476,E2 -7767.476} C_VEL
LIN {X 0,Y 620.824,Z 320.211,A -85,B 0,C 180,E1 -7770.137,E2 -7770.137} C_VEL
LIN {X 0,Y 621.248,Z 300.373,A -85,B 0,C 180,E1 -7772.617,E2 -7772.617} C_VEL
LIN {X 0,Y 621.403,Z 290.062,A -85,B 0,C 180,E1 -7773.915,E2 -7773.915} C_VEL
LIN {X 0,Y 619.64,Z 279.859,A -85,B 0,C 180,E1 -7775.283,E2 -7775.283} C_VEL
LIN {X 0,Y 619.604,Z 279.862,A -85,B 0,C 180,E1 -7777.689,E2 -7777.689} C_VEL
LIN {X 0,Y 619.586,Z 279.868,A -85,B 0,C 180,E1 -7780.12,E2 -7780.12} C_VEL
LIN {X 0,Y 619.565,Z 279.863,A -85,B 0,C 180,E1 -7781.319,E2 -7781.319} C_VEL
LIN {X 0,Y 618.903,Z 279.951,A -85,B 0,C 180,E1 -7781.862,E2 -7781.862} C_VEL
LIN {X 0,Y 616.054,Z 280.304,A -85,B 0,C 180,E1 -7782.743,E2 -7782.743} C_VEL
LIN {X 0,Y 613.652,Z 280.604,A -85,B 0,C 180,E1 -7783.452,E2 -7783.452} C_VEL
LIN {X 0,Y 612.629,Z 280.734,A -85,B 0,C 180,E1 -7783.999,E2 -7783.999} C_VEL
LIN {X 0,Y 612.551,Z 280.743,A -85,B 0,C 180,E1 -7784.184,E2 -7784.184} C_VEL
LIN {X 0,Y 612.535,Z 280.741,A -85,B 0,C 180,E1 -7787.042,E2 -7787.042} C_VEL
LIN {X 0,Y 612.54,Z 280.742,A -85,B 0,C 180,E1 -7789.321,E2 -7789.321} C_VEL
LIN {X 0,Y 612.528,Z 280.743,A -85,B 0,C 180,E1 -7792.096,E2 -7792.096} C_VEL
LIN {X 0,Y 612.572,Z 280.736,A -85,B 0,C 180,E1 -7794.326,E2 -7794.326} C_VEL
LIN {X 0,Y 612.554,Z 280.74,A -85,B 0,C 180,E1 -7796.709,E2 -7796.709} C_VEL
LIN {X 0,Y 612.552,Z 280.742,A -85,B 0,C 180,E1 -7799.05,E2 -7799.05} C_VEL
LIN {X 0,Y 612.573,Z 280.737,A -85,B 0,C 180,E1 -7801.697,E2 -7801.697} C_VEL
LIN {X 0,Y 612.556,Z 280.743,A -85,B 0,C 180,E1 -7804.602,E2 -7804.602} C_VEL
LIN {X 0,Y 612.585,Z 280.737,A -85,B 0,C 180,E1 -7807.121,E2 -7807.121} C_VEL
LIN {X 0,Y 612.607,Z 280.732,A -85,B 0,C 180,E1 -7809.938,E2 -7809.938} C_VEL
LIN {X 0,Y 612.599,Z 280.735,A -85,B 0,C 180,E1 -7812.704,E2 -7812.704} C_VEL
LIN {X 0,Y 612.628,Z 280.728,A -85,B 0,C 180,E1 -7815.43,E2 -7815.43} C_VEL
LIN {X 0,Y 612.618,Z 280.736,A -85,B 0,C 180,E1 -7818.122,E2 -7818.122} C_VEL
LIN {X 0,Y 612.6,Z 280.733,A -85,B 0,C 180,E1 -7820.787,E2 -7820.787} C_VEL
LIN {X 0,Y 612.71,Z 280.725,A -85,B 0,C 180,E1 -7823.589,E2 -7823.589} C_VEL
LIN {X 0,Y 613.527,Z 287.204,A -85,B 0,C 180,E1 -7824.758,E2 -7824.758} C_VEL
LIN {X 0,Y 613.378,Z 297.379,A -85,B 0,C 180,E1 -7826.479,E2 -7826.479} C_VEL
LIN {X 0,Y 615.948,Z 310.106,A -85,B 0,C 180,E1 -7826.698,E2 -7826.698} C_VEL
LIN {X 0,Y 615.162,Z 432.537,A -85,B 0,C 180,E1 -7828.143,E2 -7828.143} C_VEL
LIN {X 0,Y 614.988,Z 447.002,A -85,B 0,C 180,E1 -7828.448,E2 -7828.448} C_VEL
LIN {X 0,Y 614.682,Z 461.394,A -85,B 0,C 180,E1 -7828.897,E2 -7828.897} C_VEL
LIN {X 0,Y 614.368,Z 474.126,A -85,B 0,C 180,E1 -7829.427,E2 -7829.427} C_VEL
LIN {X 0,Y 614.004,Z 486.513,A -85,B 0,C 180,E1 -7830.08,E2 -7830.08} C_VEL
LIN {X 0,Y 613.567,Z 497.858,A -85,B 0,C 180,E1 -7830.816,E2 -7830.816} C_VEL
LIN {X 0,Y 613.259,Z 508.25,A -85,B 0,C 180,E1 -7831.635,E2 -7831.635} C_VEL
LIN {X 0,Y 612.786,Z 518.628,A -85,B 0,C 180,E1 -7832.619,E2 -7832.619} C_VEL
LIN {X 0,Y 612.536,Z 527.18,A -85,B 0,C 180,E1 -7833.604,E2 -7833.604} C_VEL
LIN {X 0,Y 612.184,Z 535.431,A -85,B 0,C 180,E1 -7834.757,E2 -7834.757} C_VEL
LIN {X 0,Y 612.052,Z 542.055,A -85,B 0,C 180,E1 -7835.91,E2 -7835.91} C_VEL
LIN {X 0,Y 611.874,Z 547.957,A -85,B 0,C 180,E1 -7837.232,E2 -7837.232} C_VEL
LIN {X 0,Y 611.725,Z 552.301,A -85,B 0,C 180,E1 -7838.559,E2 -7838.559} C_VEL
LIN {X 0,Y 611.685,Z 555.205,A -85,B 0,C 180,E1 -7839.889,E2 -7839.889} C_VEL
LIN {X 0,Y 611.643,Z 556.748,A -85,B 0,C 180,E1 -7841.224,E2 -7841.224} C_VEL
LIN {X 0,Y 611.665,Z 556.942,A -85,B 0,C 180,E1 -7842.565,E2 -7842.565} C_VEL
LIN {X 0,Y 611.658,Z 555.78,A -85,B 0,C 180,E1 -7843.913,E2 -7843.913} C_VEL
LIN {X 0,Y 611.741,Z 553.2,A -85,B 0,C 180,E1 -7845.267,E2 -7845.267} C_VEL
LIN {X 0,Y 611.877,Z 549.085,A -85,B 0,C 180,E1 -7846.628,E2 -7846.628} C_VEL
LIN {X 0,Y 612.003,Z 544.957,A -85,B 0,C 180,E1 -7847.654,E2 -7847.654} C_VEL
LIN {X 0,Y 612.171,Z 539.75,A -85,B 0,C 180,E1 -7848.684,E2 -7848.684} C_VEL
LIN {X 0,Y 612.458,Z 532.237,A -85,B 0,C 180,E1 -7849.889,E2 -7849.889} C_VEL
LIN {X 0,Y 612.747,Z 524.263,A -85,B 0,C 180,E1 -7850.928,E2 -7850.928} C_VEL
LIN {X 0,Y 613.187,Z 514.556,A -85,B 0,C 180,E1 -7851.967,E2 -7851.967} C_VEL
LIN {X 0,Y 613.539,Z 503.648,A -85,B 0,C 180,E1 -7852.927,E2 -7852.927} C_VEL
LIN {X 0,Y 614.035,Z 491.616,A -85,B 0,C 180,E1 -7853.788,E2 -7853.788} C_VEL
LIN {X 0,Y 614.421,Z 479.425,A -85,B 0,C 180,E1 -7854.497,E2 -7854.497} C_VEL
LIN {X 0,Y 614.827,Z 466.137,A -85,B 0,C 180,E1 -7855.109,E2 -7855.109} C_VEL
LIN {X 0,Y 615.198,Z 452.397,A -85,B 0,C 180,E1 -7855.589,E2 -7855.589} C_VEL
LIN {X 0,Y 615.355,Z 438.761,A -85,B 0,C 180,E1 -7855.93,E2 -7855.93} C_VEL
LIN {X 0,Y 615.455,Z 423.091,A -85,B 0,C 180,E1 -7856.171,E2 -7856.171} C_VEL
LIN {X 0,Y 616.197,Z 309.993,A -85,B 0,C 180,E1 -7857.504,E2 -7857.504} C_VEL
LIN {X 0,Y 613.586,Z 297.678,A -85,B 0,C 180,E1 -7857.747,E2 -7857.747} C_VEL
LIN {X 0,Y 613.756,Z 288.114,A -85,B 0,C 180,E1 -7859.386,E2 -7859.386} C_VEL
LIN {X 0,Y 612.56,Z 280.744,A -85,B 0,C 180,E1 -7860.742,E2 -7860.742} C_VEL
LIN {X 0,Y 612.532,Z 280.741,A -85,B 0,C 180,E1 -7863.408,E2 -7863.408} C_VEL
LIN {X 0,Y 612.558,Z 280.74,A -85,B 0,C 180,E1 -7865.721,E2 -7865.721} C_VEL
LIN {X 0,Y 612.518,Z 280.747,A -85,B 0,C 180,E1 -7868.132,E2 -7868.132} C_VEL
LIN {X 0,Y 612.519,Z 280.739,A -85,B 0,C 180,E1 -7870.997,E2 -7870.997} C_VEL
LIN {X 0,Y 612.531,Z 280.746,A -85,B 0,C 180,E1 -7873.911,E2 -7873.911} C_VEL
LIN {X 0,Y 612.545,Z 280.738,A -85,B 0,C 180,E1 -7876.678,E2 -7876.678} C_VEL
LIN {X 0,Y 612.55,Z 280.738,A -85,B 0,C 180,E1 -7879.323,E2 -7879.323} C_VEL
LIN {X 0,Y 612.524,Z 280.743,A -85,B 0,C 180,E1 -7882.092,E2 -7882.092} C_VEL
LIN {X 0,Y 612.577,Z 280.726,A -85,B 0,C 180,E1 -7884.327,E2 -7884.327} C_VEL
LIN {X 0,Y 612.532,Z 280.738,A -85,B 0,C 180,E1 -7886.709,E2 -7886.709} C_VEL
LIN {X 0,Y 612.569,Z 280.732,A -85,B 0,C 180,E1 -7889.042,E2 -7889.042} C_VEL
LIN {X 0,Y 612.574,Z 280.739,A -85,B 0,C 180,E1 -7891.692,E2 -7891.692} C_VEL
LIN {X 0,Y 612.528,Z 280.739,A -85,B 0,C 180,E1 -7894.601,E2 -7894.601} C_VEL
LIN {X 0,Y 612.567,Z 280.733,A -85,B 0,C 180,E1 -7897.122,E2 -7897.122} C_VEL
LIN {X 0,Y 612.576,Z 280.733,A -85,B 0,C 180,E1 -7899.938,E2 -7899.938} C_VEL
LIN {X 0,Y 612.561,Z 280.734,A -85,B 0,C 180,E1 -7902.704,E2 -7902.704} C_VEL
LIN {X 0,Y 612.579,Z 280.732,A -85,B 0,C 180,E1 -7904.752,E2 -7904.752} C_VEL
LIN {X 0,Y 612.637,Z 280.722,A -85,B 0,C 180,E1 -7906.781,E2 -7906.781} C_VEL
LIN {X 0,Y 612.597,Z 280.734,A -85,B 0,C 180,E1 -7909.508,E2 -7909.508} C_VEL
LIN {X 0,Y 612.651,Z 280.721,A -85,B 0,C 180,E1 -7912.114,E2 -7912.114} C_VEL
LIN {X 0,Y 612.659,Z 280.725,A -85,B 0,C 180,E1 -7914.752,E2 -7914.752} C_VEL
LIN {X 0,Y 612.521,Z 280.736,A -85,B 0,C 180,E1 -7916.722,E2 -7916.722} C_VEL
LIN {X 0,Y 612.809,Z 280.709,A -85,B 0,C 180,E1 -7919.345,E2 -7919.345} C_VEL
LIN {X 0,Y 612.81,Z 280.702,A -85,B 0,C 180,E1 -7921.31,E2 -7921.31} C_VEL
LIN {X 0,Y 612.698,Z 280.72,A -85,B 0,C 180,E1 -7924.59,E2 -7924.59} C_VEL
LIN {X 0,Y 612.649,Z 280.724,A -85,B 0,C 180,E1 -7927.225,E2 -7927.225} C_VEL
LIN {X 0,Y 612.692,Z 280.721,A -85,B 0,C 180,E1 -7930.54,E2 -7930.54} C_VEL
LIN {X 0,Y 612.609,Z 280.725,A -85,B 0,C 180,E1 -7933.893,E2 -7933.893} C_VEL
LIN {X 0,Y 612.588,Z 280.736,A -85,B 0,C 180,E1 -7936.61,E2 -7936.61} C_VEL
LIN {X 0,Y 612.572,Z 280.733,A -85,B 0,C 180,E1 -7939.366,E2 -7939.366} C_VEL
LIN {X 0,Y 612.569,Z 280.732,A -85,B 0,C 180,E1 -7942.169,E2 -7942.169} C_VEL
LIN {X 0,Y 612.568,Z 280.737,A -85,B 0,C 180,E1 -7944.308,E2 -7944.308} C_VEL
LIN {X 0,Y 612.531,Z 280.738,A -85,B 0,C 180,E1 -7947.22,E2 -7947.22} C_VEL
LIN {X 0,Y 612.566,Z 280.733,A -85,B 0,C 180,E1 -7949.659,E2 -7949.659} C_VEL
LIN {X 0,Y 612.551,Z 280.744,A -85,B 0,C 180,E1 -7952.51,E2 -7952.51} C_VEL
LIN {X 0,Y 612.589,Z 280.722,A -85,B 0,C 180,E1 -7954.87,E2 -7954.87} C_VEL
LIN {X 0,Y 612.595,Z 280.727,A -85,B 0,C 180,E1 -7957.301,E2 -7957.301} C_VEL
LIN {X 0,Y 612.554,Z 280.74,A -85,B 0,C 180,E1 -7959.996,E2 -7959.996} C_VEL
LIN {X 0,Y 612.554,Z 280.741,A -85,B 0,C 180,E1 -7962.427,E2 -7962.427} C_VEL
LIN {X 0,Y 612.526,Z 280.737,A -85,B 0,C 180,E1 -7965.153,E2 -7965.153} C_VEL
LIN {X 0,Y 612.583,Z 280.733,A -85,B 0,C 180,E1 -7967.578,E2 -7967.578} C_VEL
LIN {X 0,Y 612.545,Z 280.746,A -85,B 0,C 180,E1 -7970.184,E2 -7970.184} C_VEL
LIN {X 0,Y 612.606,Z 280.729,A -85,B 0,C 180,E1 -7973.165,E2 -7973.165} C_VEL
LIN {X 0,Y 612.56,Z 280.743,A -85,B 0,C 180,E1 -7975.926,E2 -7975.926} C_VEL
LIN {X 0,Y 612.562,Z 280.745,A -85,B 0,C 180,E1 -7978.267,E2 -7978.267} C_VEL
LIN {X 0,Y 612.616,Z 280.733,A -85,B 0,C 180,E1 -7980.553,E2 -7980.553} C_VEL
LIN {X 0,Y 612.547,Z 280.741,A -85,B 0,C 180,E1 -7983.116,E2 -7983.116} C_VEL
LIN {X 0,Y 612.543,Z 280.798,A -85,B 0,C 180,E1 -7984.042,E2 -7984.042} C_VEL
LIN {X 0,Y 615.31,Z 293.831,A -85,B 0,C 180,E1 -7985.809,E2 -7985.809} C_VEL
LIN {X 0,Y 615.311,Z 300.965,A -85,B 0,C 180,E1 -7986.7,E2 -7986.7} C_VEL
LIN {X 0,Y 614.433,Z 322.353,A -85,B 0,C 180,E1 -7989.307,E2 -7989.307} C_VEL
LIN {X 0,Y 613.712,Z 343.762,A -85,B 0,C 180,E1 -7991.882,E2 -7991.882} C_VEL
LIN {X 0,Y 613.17,Z 364.066,A -85,B 0,C 180,E1 -7994.291,E2 -7994.291} C_VEL
LIN {X 0,Y 615.935,Z 385.809,A -85,B 0,C 180,E1 -7994.628,E2 -7994.628} C_VEL
LIN {X 0,Y 615.19,Z 502.738,A -85,B 0,C 180,E1 -7996.021,E2 -7996.021} C_VEL
LIN {X 0,Y 614.826,Z 517.166,A -85,B 0,C 180,E1 -7996.328,E2 -7996.328} C_VEL
LIN {X 0,Y 614.423,Z 530.474,A -85,B 0,C 180,E1 -7996.739,E2 -7996.739} C_VEL
LIN {X 0,Y 613.942,Z 544.428,A -85,B 0,C 180,E1 -7997.315,E2 -7997.315} C_VEL
LIN {X 0,Y 613.481,Z 556.931,A -85,B 0,C 180,E1 -7997.975,E2 -7997.975} C_VEL
LIN {X 0,Y 613.062,Z 568.367,A -85,B 0,C 180,E1 -7998.719,E2 -7998.719} C_VEL
LIN {X 0,Y 612.746,Z 579.452,A -85,B 0,C 180,E1 -7999.593,E2 -7999.593} C_VEL
LIN {X 0,Y 612.392,Z 588.567,A -85,B 0,C 180,E1 -8000.455,E2 -8000.455} C_VEL
LIN {X 0,Y 612.052,Z 597.372,A -85,B 0,C 180,E1 -8001.446,E2 -8001.446} C_VEL
LIN {X 0,Y 611.85,Z 605.84,A -85,B 0,C 180,E1 -8002.602,E2 -8002.602} C_VEL
LIN {X 0,Y 611.729,Z 612.697,A -85,B 0,C 180,E1 -8003.757,E2 -8003.757} C_VEL
LIN {X 0,Y 611.632,Z 619.13,A -85,B 0,C 180,E1 -8005.09,E2 -8005.09} C_VEL
LIN {X 0,Y 611.648,Z 622.706,A -85,B 0,C 180,E1 -8006.062,E2 -8006.062} C_VEL
LIN {X 0,Y 611.602,Z 626.242,A -85,B 0,C 180,E1 -8007.376,E2 -8007.376} C_VEL
LIN {X 0,Y 611.643,Z 628.34,A -85,B 0,C 180,E1 -8008.689,E2 -8008.689} C_VEL
LIN {X 0,Y 611.632,Z 629.039,A -85,B 0,C 180,E1 -8010.002,E2 -8010.002} C_VEL
LIN {X 0,Y 611.644,Z 628.336,A -85,B 0,C 180,E1 -8011.314,E2 -8011.314} C_VEL
LIN {X 0,Y 611.605,Z 626.23,A -85,B 0,C 180,E1 -8012.627,E2 -8012.627} C_VEL
LIN {X 0,Y 611.649,Z 622.68,A -85,B 0,C 180,E1 -8013.941,E2 -8013.941} C_VEL
LIN {X 0,Y 611.654,Z 617.585,A -85,B 0,C 180,E1 -8015.258,E2 -8015.258} C_VEL
LIN {X 0,Y 611.727,Z 612.637,A -85,B 0,C 180,E1 -8016.246,E2 -8016.246} C_VEL
LIN {X 0,Y 611.869,Z 604.534,A -85,B 0,C 180,E1 -8017.566,E2 -8017.566} C_VEL
LIN {X 0,Y 612.12,Z 595.749,A -85,B 0,C 180,E1 -8018.722,E2 -8018.722} C_VEL
LIN {X 0,Y 612.38,Z 586.557,A -85,B 0,C 180,E1 -8019.714,E2 -8019.714} C_VEL
LIN {X 0,Y 612.722,Z 577.404,A -85,B 0,C 180,E1 -8020.541,E2 -8020.541} C_VEL
LIN {X 0,Y 613.073,Z 566.485,A -85,B 0,C 180,E1 -8021.368,E2 -8021.368} C_VEL
LIN {X 0,Y 613.462,Z 554.541,A -85,B 0,C 180,E1 -8022.112,E2 -8022.112} C_VEL
LIN {X 0,Y 613.96,Z 541.357,A -85,B 0,C 180,E1 -8022.772,E2 -8022.772} C_VEL
LIN {X 0,Y 614.353,Z 527.395,A -85,B 0,C 180,E1 -8023.308,E2 -8023.308} C_VEL
LIN {X 0,Y 614.721,Z 513.467,A -85,B 0,C 180,E1 -8023.699,E2 -8023.699} C_VEL
LIN {X 0,Y 615.006,Z 499.005,A -85,B 0,C 180,E1 -8023.965,E2 -8023.965} C_VEL
LIN {X 0,Y 615.615,Z 384.439,A -85,B 0,C 180,E1 -8025.309,E2 -8025.309} C_VEL
LIN {X 0,Y 613.097,Z 364.247,A -85,B 0,C 180,E1 -8025.618,E2 -8025.618} C_VEL
LIN {X 0,Y 613.779,Z 337.234,A -85,B 0,C 180,E1 -8028.791,E2 -8028.791} C_VEL
LIN {X 0,Y 614.507,Z 313.812,A -85,B 0,C 180,E1 -8031.569,E2 -8031.569} C_VEL
LIN {X 0,Y 615.196,Z 294.872,A -85,B 0,C 180,E1 -8033.842,E2 -8033.842} C_VEL
LIN {X 0,Y 613.955,Z 287.438,A -85,B 0,C 180,E1 -8034.79,E2 -8034.79} C_VEL
LIN {X 0,Y 612.559,Z 280.743,A -85,B 0,C 180,E1 -8035.683,E2 -8035.683} C_VEL
LIN {X 0,Y 612.573,Z 280.739,A -85,B 0,C 180,E1 -8038.303,E2 -8038.303} C_VEL
LIN {X 0,Y 612.546,Z 280.738,A -85,B 0,C 180,E1 -8040.97,E2 -8040.97} C_VEL
LIN {X 0,Y 612.548,Z 280.741,A -85,B 0,C 180,E1 -8043.41,E2 -8043.41} C_VEL
LIN {X 0,Y 612.554,Z 280.744,A -85,B 0,C 180,E1 -8045.721,E2 -8045.721} C_VEL
LIN {X 0,Y 612.529,Z 280.741,A -85,B 0,C 180,E1 -8048.135,E2 -8048.135} C_VEL
LIN {X 0,Y 612.539,Z 280.743,A -85,B 0,C 180,E1 -8050.999,E2 -8050.999} C_VEL
LIN {X 0,Y 612.544,Z 280.738,A -85,B 0,C 180,E1 -8053.912,E2 -8053.912} C_VEL
LIN {X 0,Y 612.559,Z 280.739,A -85,B 0,C 180,E1 -8056.679,E2 -8056.679} C_VEL
